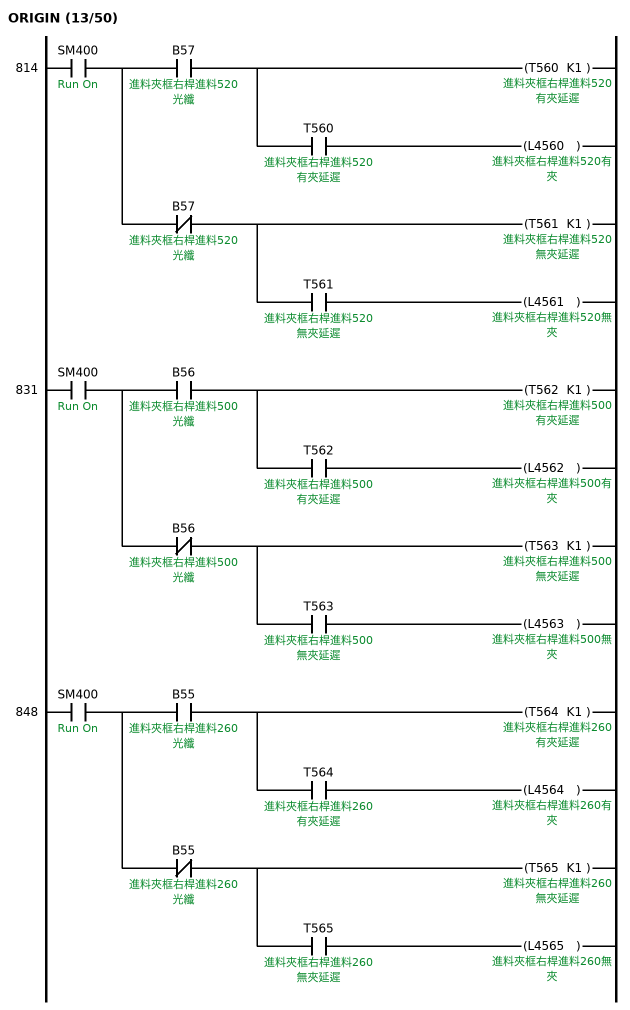
[picture p432: ladder of ORIGIN, rungs at steps 814 to 848]
814   LD      SM400  ; Run On
      MPS
      AND     B57  ; 進料夾框右桿進料520 光纖
      OUT     T560 K1  ; 進料夾框右桿進料520 有夾延遲
      AND     T560  ; 進料夾框右桿進料520 有夾延遲
      OUT     L4560  ; 進料夾框右桿進料520有夾
      MPP
      ANI     B57  ; 進料夾框右桿進料520 光纖
      OUT     T561 K1  ; 進料夾框右桿進料520 無夾延遲
      AND     T561  ; 進料夾框右桿進料520 無夾延遲
      OUT     L4561  ; 進料夾框右桿進料520無夾
831   LD      SM400  ; Run On
      MPS
      AND     B56  ; 進料夾框右桿進料500 光纖
      OUT     T562 K1  ; 進料夾框右桿進料500 有夾延遲
      AND     T562  ; 進料夾框右桿進料500 有夾延遲
      OUT     L4562  ; 進料夾框右桿進料500有夾
      MPP
      ANI     B56  ; 進料夾框右桿進料500 光纖
      OUT     T563 K1  ; 進料夾框右桿進料500 無夾延遲
      AND     T563  ; 進料夾框右桿進料500 無夾延遲
      OUT     L4563  ; 進料夾框右桿進料500無夾
848   LD      SM400  ; Run On
      MPS
      AND     B55  ; 進料夾框右桿進料260 光纖
      OUT     T564 K1  ; 進料夾框右桿進料260 有夾延遲
      AND     T564  ; 進料夾框右桿進料260 有夾延遲
      OUT     L4564  ; 進料夾框右桿進料260有夾
      MPP
      ANI     B55  ; 進料夾框右桿進料260 光纖
      OUT     T565 K1  ; 進料夾框右桿進料260 無夾延遲
      AND     T565  ; 進料夾框右桿進料260 無夾延遲
      OUT     L4565  ; 進料夾框右桿進料260無夾
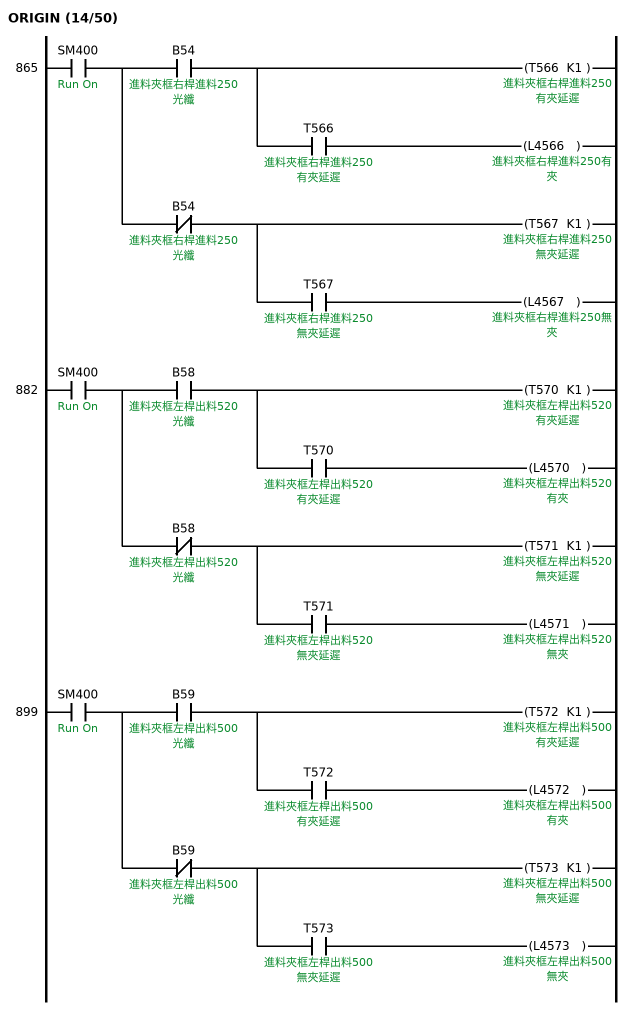
865   LD      SM400  ; Run On
      MPS
      AND     B54  ; 進料夾框右桿進料250 光纖
      OUT     T566 K1  ; 進料夾框右桿進料250 有夾延遲
      AND     T566  ; 進料夾框右桿進料250 有夾延遲
      OUT     L4566  ; 進料夾框右桿進料250有夾
      MPP
      ANI     B54  ; 進料夾框右桿進料250 光纖
      OUT     T567 K1  ; 進料夾框右桿進料250 無夾延遲
      AND     T567  ; 進料夾框右桿進料250 無夾延遲
      OUT     L4567  ; 進料夾框右桿進料250無夾
882   LD      SM400  ; Run On
      MPS
      AND     B58  ; 進料夾框左桿出料520 光纖
      OUT     T570 K1  ; 進料夾框左桿出料520 有夾延遲
      AND     T570  ; 進料夾框左桿出料520 有夾延遲
      OUT     L4570  ; 進料夾框左桿出料520 有夾
      MPP
      ANI     B58  ; 進料夾框左桿出料520 光纖
      OUT     T571 K1  ; 進料夾框左桿出料520 無夾延遲
      AND     T571  ; 進料夾框左桿出料520 無夾延遲
      OUT     L4571  ; 進料夾框左桿出料520 無夾
899   LD      SM400  ; Run On
      MPS
      AND     B59  ; 進料夾框左桿出料500 光纖
      OUT     T572 K1  ; 進料夾框左桿出料500 有夾延遲
      AND     T572  ; 進料夾框左桿出料500 有夾延遲
      OUT     L4572  ; 進料夾框左桿出料500 有夾
      MPP
      ANI     B59  ; 進料夾框左桿出料500 光纖
      OUT     T573 K1  ; 進料夾框左桿出料500 無夾延遲
      AND     T573  ; 進料夾框左桿出料500 無夾延遲
      OUT     L4573  ; 進料夾框左桿出料500 無夾
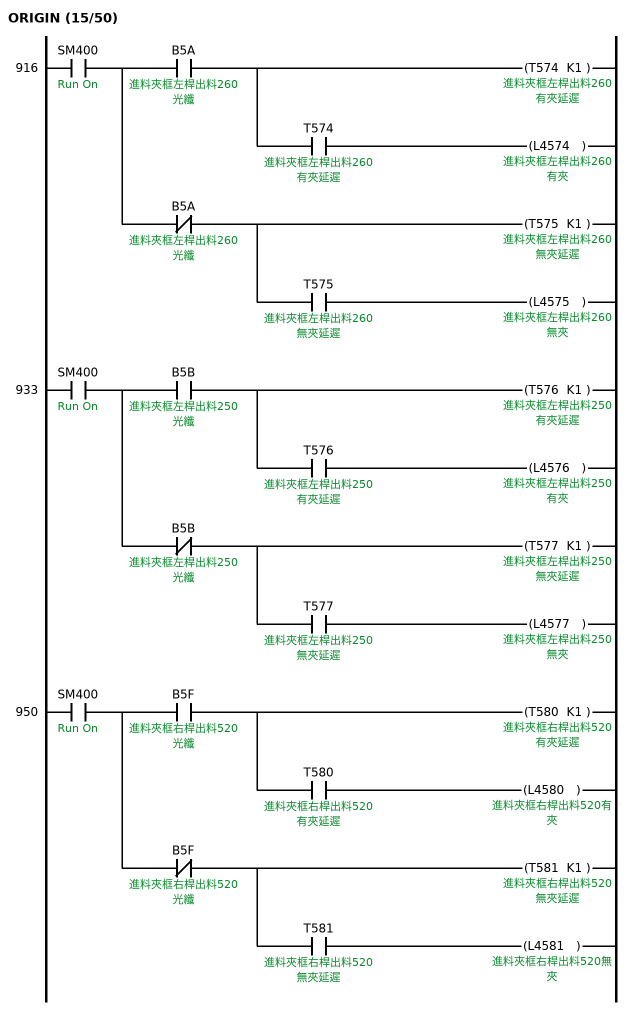
916   LD      SM400  ; Run On
      MPS
      AND     B5A  ; 進料夾框左桿出料260 光纖
      OUT     T574 K1  ; 進料夾框左桿出料260 有夾延遲
      AND     T574  ; 進料夾框左桿出料260 有夾延遲
      OUT     L4574  ; 進料夾框左桿出料260 有夾
      MPP
      ANI     B5A  ; 進料夾框左桿出料260 光纖
      OUT     T575 K1  ; 進料夾框左桿出料260 無夾延遲
      AND     T575  ; 進料夾框左桿出料260 無夾延遲
      OUT     L4575  ; 進料夾框左桿出料260 無夾
933   LD      SM400  ; Run On
      MPS
      AND     B5B  ; 進料夾框左桿出料250 光纖
      OUT     T576 K1  ; 進料夾框左桿出料250 有夾延遲
      AND     T576  ; 進料夾框左桿出料250 有夾延遲
      OUT     L4576  ; 進料夾框左桿出料250 有夾
      MPP
      ANI     B5B  ; 進料夾框左桿出料250 光纖
      OUT     T577 K1  ; 進料夾框左桿出料250 無夾延遲
      AND     T577  ; 進料夾框左桿出料250 無夾延遲
      OUT     L4577  ; 進料夾框左桿出料250 無夾
950   LD      SM400  ; Run On
      MPS
      AND     B5F  ; 進料夾框右桿出料520 光纖
      OUT     T580 K1  ; 進料夾框右桿出料520 有夾延遲
      AND     T580  ; 進料夾框右桿出料520 有夾延遲
      OUT     L4580  ; 進料夾框右桿出料520有夾
      MPP
      ANI     B5F  ; 進料夾框右桿出料520 光纖
      OUT     T581 K1  ; 進料夾框右桿出料520 無夾延遲
      AND     T581  ; 進料夾框右桿出料520 無夾延遲
      OUT     L4581  ; 進料夾框右桿出料520無夾
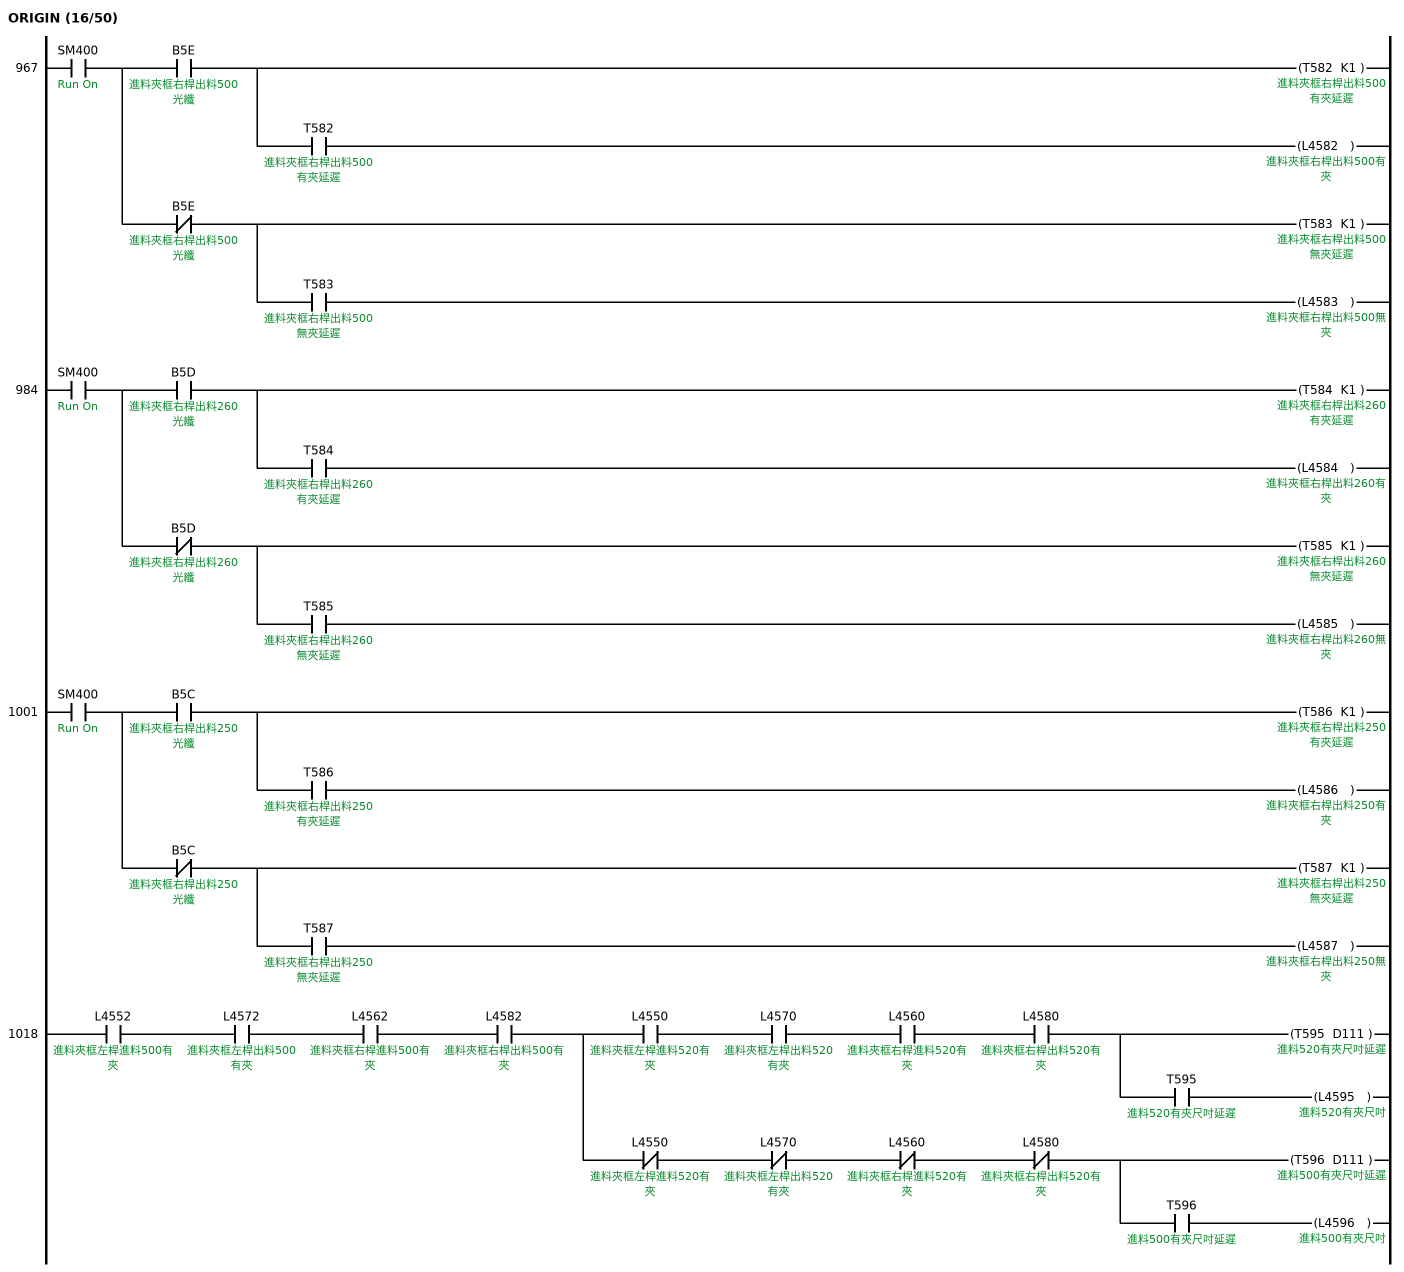
967   LD      SM400  ; Run On
      MPS
      AND     B5E  ; 進料夾框右桿出料500 光纖
      OUT     T582 K1  ; 進料夾框右桿出料500 有夾延遲
      AND     T582  ; 進料夾框右桿出料500 有夾延遲
      OUT     L4582  ; 進料夾框右桿出料500有夾
      MPP
      ANI     B5E  ; 進料夾框右桿出料500 光纖
      OUT     T583 K1  ; 進料夾框右桿出料500 無夾延遲
      AND     T583  ; 進料夾框右桿出料500 無夾延遲
      OUT     L4583  ; 進料夾框右桿出料500無夾
984   LD      SM400  ; Run On
      MPS
      AND     B5D  ; 進料夾框右桿出料260 光纖
      OUT     T584 K1  ; 進料夾框右桿出料260 有夾延遲
      AND     T584  ; 進料夾框右桿出料260 有夾延遲
      OUT     L4584  ; 進料夾框右桿出料260有夾
      MPP
      ANI     B5D  ; 進料夾框右桿出料260 光纖
      OUT     T585 K1  ; 進料夾框右桿出料260 無夾延遲
      AND     T585  ; 進料夾框右桿出料260 無夾延遲
      OUT     L4585  ; 進料夾框右桿出料260無夾
1001  LD      SM400  ; Run On
      MPS
      AND     B5C  ; 進料夾框右桿出料250 光纖
      OUT     T586 K1  ; 進料夾框右桿出料250 有夾延遲
      AND     T586  ; 進料夾框右桿出料250 有夾延遲
      OUT     L4586  ; 進料夾框右桿出料250有夾
      MPP
      ANI     B5C  ; 進料夾框右桿出料250 光纖
      OUT     T587 K1  ; 進料夾框右桿出料250 無夾延遲
      AND     T587  ; 進料夾框右桿出料250 無夾延遲
      OUT     L4587  ; 進料夾框右桿出料250無夾
1018  LD      L4552  ; 進料夾框左桿進料500有夾
      AND     L4572  ; 進料夾框左桿出料500 有夾
      AND     L4562  ; 進料夾框右桿進料500有夾
      AND     L4582  ; 進料夾框右桿出料500有夾
      MPS
      AND     L4550  ; 進料夾框左桿進料520有夾
      AND     L4570  ; 進料夾框左桿出料520 有夾
      AND     L4560  ; 進料夾框右桿進料520有夾
      AND     L4580  ; 進料夾框右桿出料520有夾
      OUT     T595 D111  ; 進料520有夾尺吋延遲
      AND     T595  ; 進料520有夾尺吋延遲
      OUT     L4595  ; 進料520有夾尺吋
      MPP
      ANI     L4550  ; 進料夾框左桿進料520有夾
      ANI     L4570  ; 進料夾框左桿出料520 有夾
      ANI     L4560  ; 進料夾框右桿進料520有夾
      ANI     L4580  ; 進料夾框右桿出料520有夾
      OUT     T596 D111  ; 進料500有夾尺吋延遲
      AND     T596  ; 進料500有夾尺吋延遲
      OUT     L4596  ; 進料500有夾尺吋
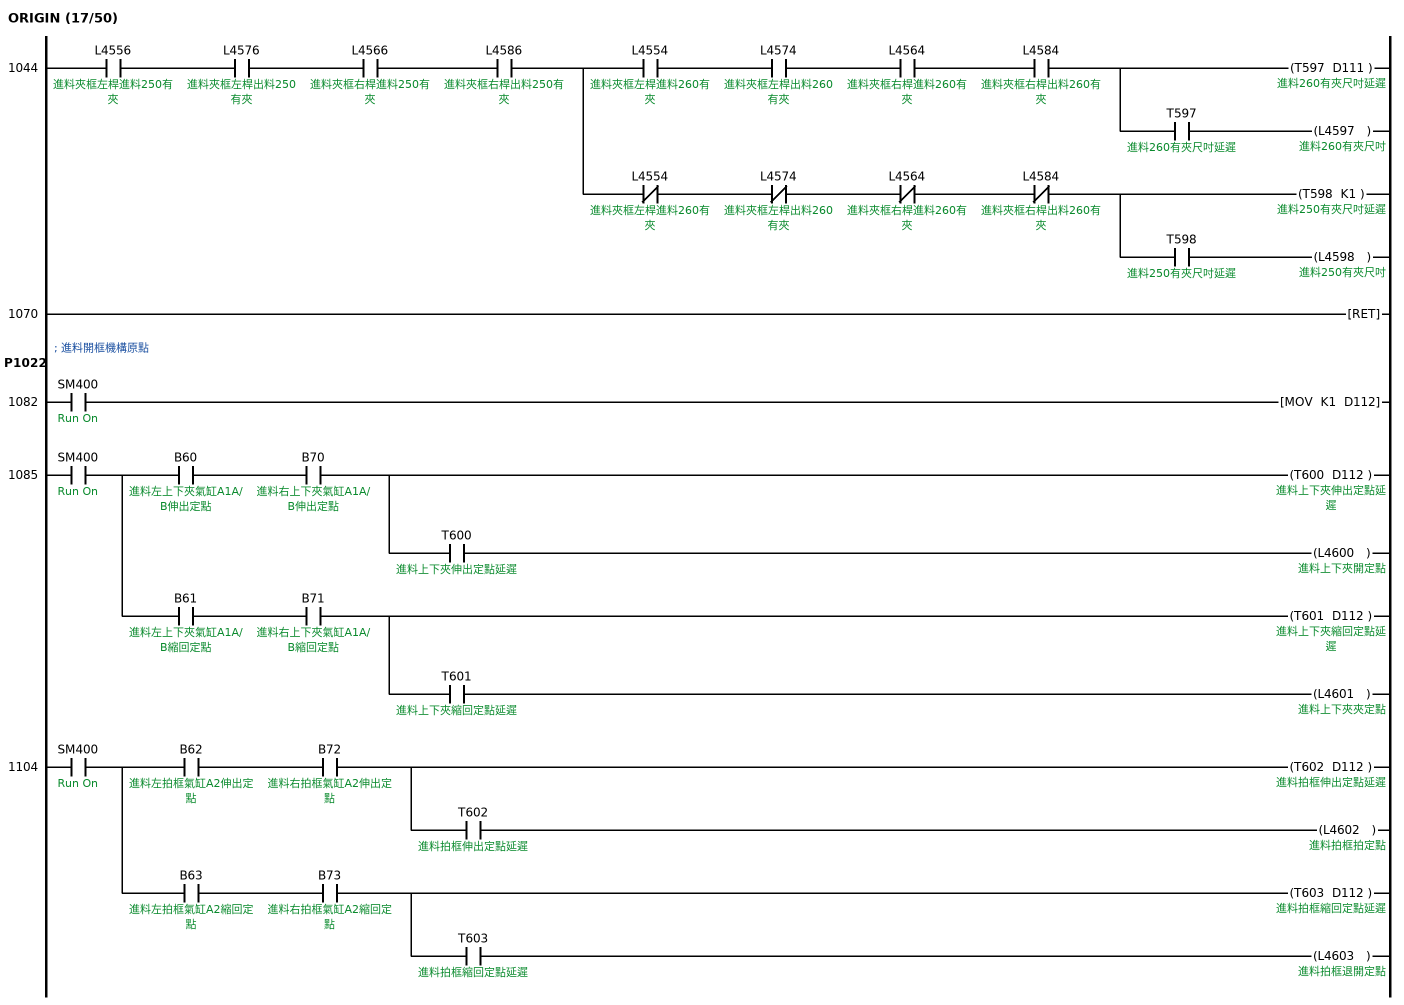
1044  LD      L4556  ; 進料夾框左桿進料250有夾
      AND     L4576  ; 進料夾框左桿出料250 有夾
      AND     L4566  ; 進料夾框右桿進料250有夾
      AND     L4586  ; 進料夾框右桿出料250有夾
      MPS
      AND     L4554  ; 進料夾框左桿進料260有夾
      AND     L4574  ; 進料夾框左桿出料260 有夾
      AND     L4564  ; 進料夾框右桿進料260有夾
      AND     L4584  ; 進料夾框右桿出料260有夾
      OUT     T597 D111  ; 進料260有夾尺吋延遲
      AND     T597  ; 進料260有夾尺吋延遲
      OUT     L4597  ; 進料260有夾尺吋
      MPP
      ANI     L4554  ; 進料夾框左桿進料260有夾
      ANI     L4574  ; 進料夾框左桿出料260 有夾
      ANI     L4564  ; 進料夾框右桿進料260有夾
      ANI     L4584  ; 進料夾框右桿出料260有夾
      OUT     T598 K1  ; 進料250有夾尺吋延遲
      AND     T598  ; 進料250有夾尺吋延遲
      OUT     L4598  ; 進料250有夾尺吋
1070  RET
; 進料開框機構原點
      P1022
1082  LD      SM400  ; Run On
      MOV     K1 D112
1085  LD      SM400  ; Run On
      MPS
      AND     B60  ; 進料左上下夾氣缸A1A/B伸出定點
      AND     B70  ; 進料右上下夾氣缸A1A/B伸出定點
      OUT     T600 D112  ; 進料上下夾伸出定點延遲
      AND     T600  ; 進料上下夾伸出定點延遲
      OUT     L4600  ; 進料上下夾開定點
      MPP
      AND     B61  ; 進料左上下夾氣缸A1A/B縮回定點
      AND     B71  ; 進料右上下夾氣缸A1A/B縮回定點
      OUT     T601 D112  ; 進料上下夾縮回定點延遲
      AND     T601  ; 進料上下夾縮回定點延遲
      OUT     L4601  ; 進料上下夾夾定點
1104  LD      SM400  ; Run On
      MPS
      AND     B62  ; 進料左拍框氣缸A2伸出定點
      AND     B72  ; 進料右拍框氣缸A2伸出定點
      OUT     T602 D112  ; 進料拍框伸出定點延遲
      AND     T602  ; 進料拍框伸出定點延遲
      OUT     L4602  ; 進料拍框拍定點
      MPP
      AND     B63  ; 進料左拍框氣缸A2縮回定點
      AND     B73  ; 進料右拍框氣缸A2縮回定點
      OUT     T603 D112  ; 進料拍框縮回定點延遲
      AND     T603  ; 進料拍框縮回定點延遲
      OUT     L4603  ; 進料拍框退開定點
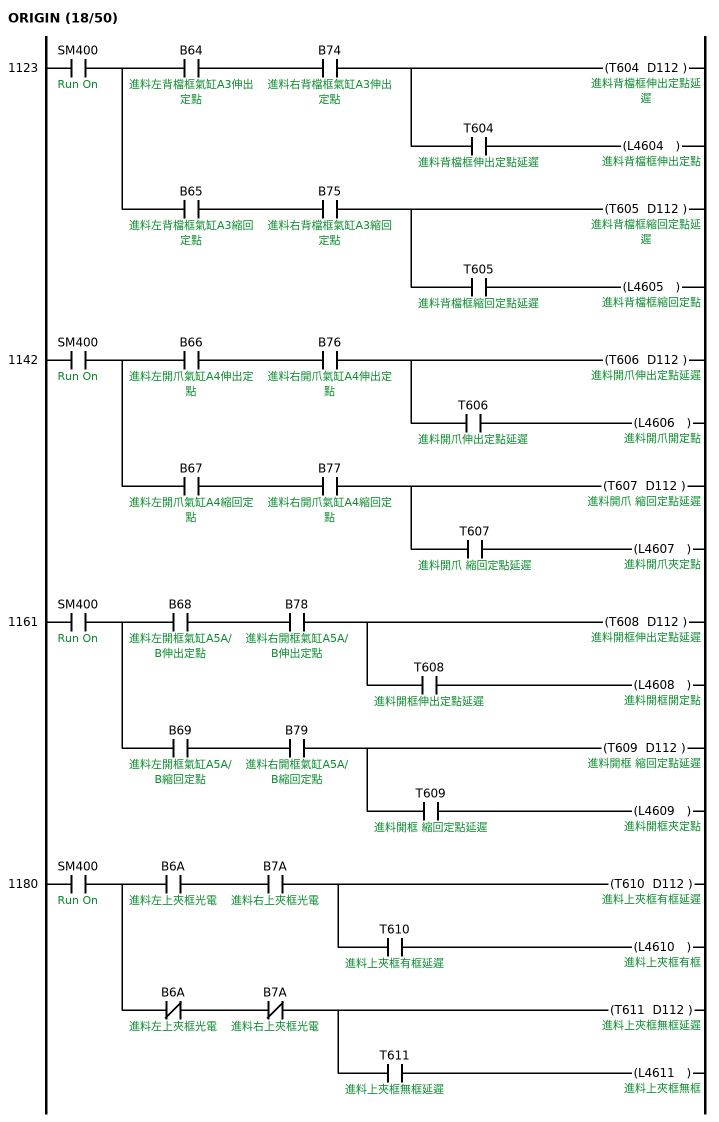
1123  LD      SM400  ; Run On
      MPS
      AND     B64  ; 進料左背檔框氣缸A3伸出定點
      AND     B74  ; 進料右背檔框氣缸A3伸出定點
      OUT     T604 D112  ; 進料背檔框伸出定點延遲
      AND     T604  ; 進料背檔框伸出定點延遲
      OUT     L4604  ; 進料背檔框伸出定點
      MPP
      AND     B65  ; 進料左背檔框氣缸A3縮回定點
      AND     B75  ; 進料右背檔框氣缸A3縮回定點
      OUT     T605 D112  ; 進料背檔框縮回定點延遲
      AND     T605  ; 進料背檔框縮回定點延遲
      OUT     L4605  ; 進料背檔框縮回定點
1142  LD      SM400  ; Run On
      MPS
      AND     B66  ; 進料左開爪氣缸A4伸出定點
      AND     B76  ; 進料右開爪氣缸A4伸出定點
      OUT     T606 D112  ; 進料開爪伸出定點延遲
      AND     T606  ; 進料開爪伸出定點延遲
      OUT     L4606  ; 進料開爪開定點
      MPP
      AND     B67  ; 進料左開爪氣缸A4縮回定點
      AND     B77  ; 進料右開爪氣缸A4縮回定點
      OUT     T607 D112  ; 進料開爪 縮回定點延遲
      AND     T607  ; 進料開爪 縮回定點延遲
      OUT     L4607  ; 進料開爪夾定點
1161  LD      SM400  ; Run On
      MPS
      AND     B68  ; 進料左開框氣缸A5A/B伸出定點
      AND     B78  ; 進料右開框氣缸A5A/B伸出定點
      OUT     T608 D112  ; 進料開框伸出定點延遲
      AND     T608  ; 進料開框伸出定點延遲
      OUT     L4608  ; 進料開框開定點
      MPP
      AND     B69  ; 進料左開框氣缸A5A/B縮回定點
      AND     B79  ; 進料右開框氣缸A5A/B縮回定點
      OUT     T609 D112  ; 進料開框 縮回定點延遲
      AND     T609  ; 進料開框 縮回定點延遲
      OUT     L4609  ; 進料開框夾定點
1180  LD      SM400  ; Run On
      MPS
      AND     B6A  ; 進料左上夾框光電
      AND     B7A  ; 進料右上夾框光電
      OUT     T610 D112  ; 進料上夾框有框延遲
      AND     T610  ; 進料上夾框有框延遲
      OUT     L4610  ; 進料上夾框有框
      MPP
      ANI     B6A  ; 進料左上夾框光電
      ANI     B7A  ; 進料右上夾框光電
      OUT     T611 D112  ; 進料上夾框無框延遲
      AND     T611  ; 進料上夾框無框延遲
      OUT     L4611  ; 進料上夾框無框
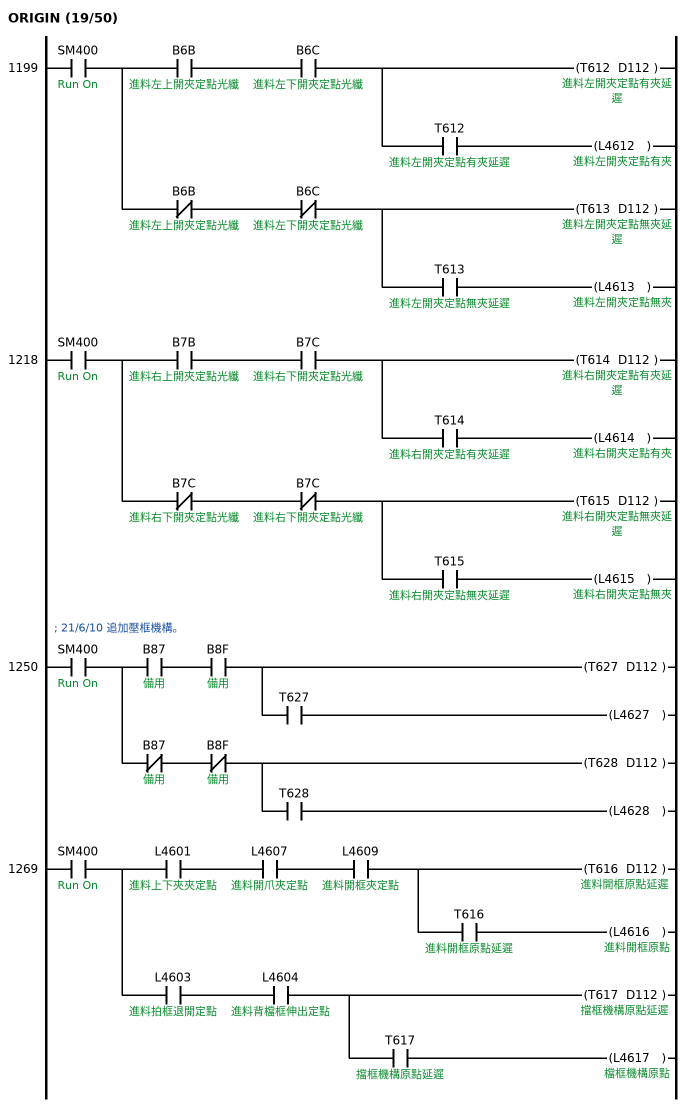
1199  LD      SM400  ; Run On
      MPS
      AND     B6B  ; 進料左上開夾定點光纖
      AND     B6C  ; 進料左下開夾定點光纖
      OUT     T612 D112  ; 進料左開夾定點有夾延遲
      AND     T612  ; 進料左開夾定點有夾延遲
      OUT     L4612  ; 進料左開夾定點有夾
      MPP
      ANI     B6B  ; 進料左上開夾定點光纖
      ANI     B6C  ; 進料左下開夾定點光纖
      OUT     T613 D112  ; 進料左開夾定點無夾延遲
      AND     T613  ; 進料左開夾定點無夾延遲
      OUT     L4613  ; 進料左開夾定點無夾
1218  LD      SM400  ; Run On
      MPS
      AND     B7B  ; 進料右上開夾定點光纖
      AND     B7C  ; 進料右下開夾定點光纖
      OUT     T614 D112  ; 進料右開夾定點有夾延遲
      AND     T614  ; 進料右開夾定點有夾延遲
      OUT     L4614  ; 進料右開夾定點有夾
      MPP
      ANI     B7C  ; 進料右下開夾定點光纖
      ANI     B7C  ; 進料右下開夾定點光纖
      OUT     T615 D112  ; 進料右開夾定點無夾延遲
      AND     T615  ; 進料右開夾定點無夾延遲
      OUT     L4615  ; 進料右開夾定點無夾
; 21/6/10 追加壓框機構。
1250  LD      SM400  ; Run On
      MPS
      AND     B87  ; 備用
      AND     B8F  ; 備用
      OUT     T627 D112
      AND     T627
      OUT     L4627
      MPP
      ANI     B87  ; 備用
      ANI     B8F  ; 備用
      OUT     T628 D112
      AND     T628
      OUT     L4628
1269  LD      SM400  ; Run On
      MPS
      AND     L4601  ; 進料上下夾夾定點
      AND     L4607  ; 進料開爪夾定點
      AND     L4609  ; 進料開框夾定點
      OUT     T616 D112  ; 進料開框原點延遲
      AND     T616  ; 進料開框原點延遲
      OUT     L4616  ; 進料開框原點
      MPP
      AND     L4603  ; 進料拍框退開定點
      AND     L4604  ; 進料背檔框伸出定點
      OUT     T617 D112  ; 擋框機構原點延遲
      AND     T617  ; 擋框機構原點延遲
      OUT     L4617  ; 檔框機構原點
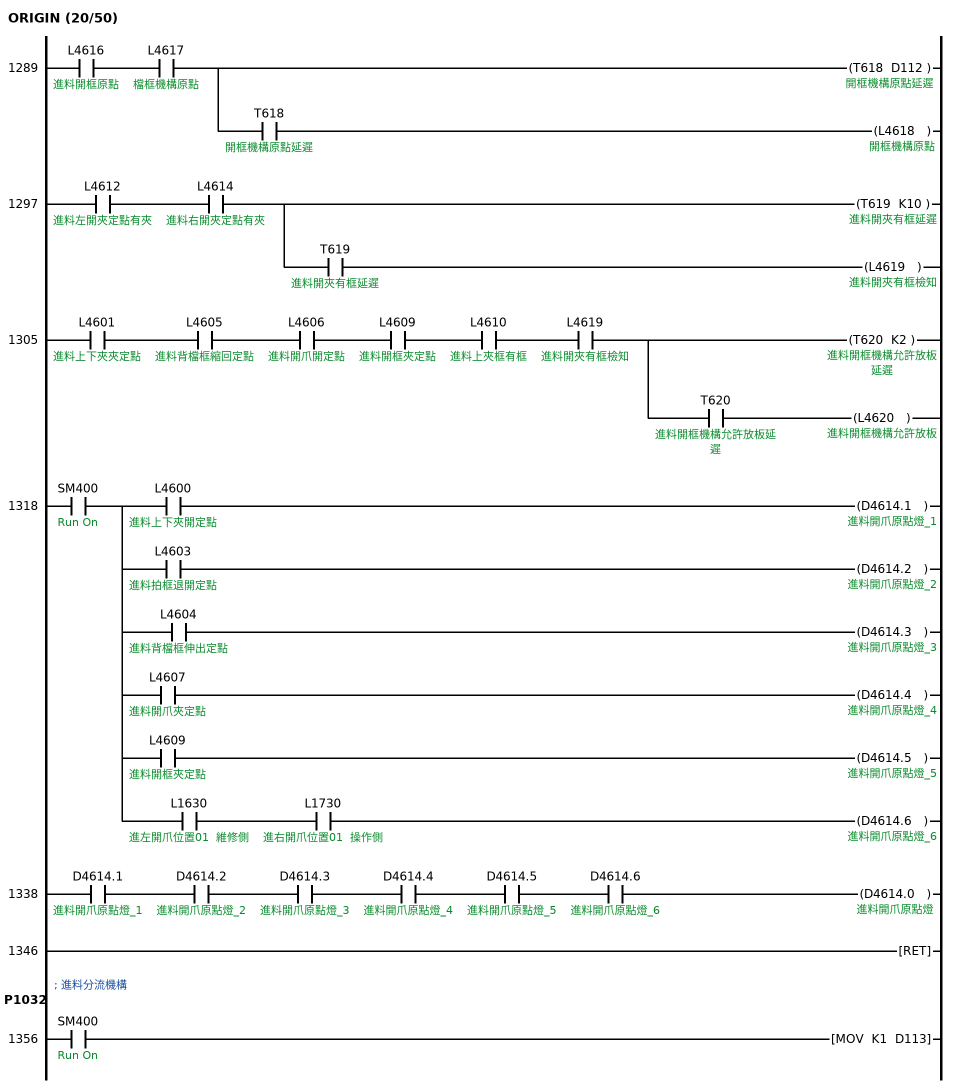
1289  LD      L4616  ; 進料開框原點
      AND     L4617  ; 檔框機構原點
      OUT     T618 D112  ; 開框機構原點延遲
      AND     T618  ; 開框機構原點延遲
      OUT     L4618  ; 開框機構原點
1297  LD      L4612  ; 進料左開夾定點有夾
      AND     L4614  ; 進料右開夾定點有夾
      OUT     T619 K10  ; 進料開夾有框延遲
      AND     T619  ; 進料開夾有框延遲
      OUT     L4619  ; 進料開夾有框檢知
1305  LD      L4601  ; 進料上下夾夾定點
      AND     L4605  ; 進料背檔框縮回定點
      AND     L4606  ; 進料開爪開定點
      AND     L4609  ; 進料開框夾定點
      AND     L4610  ; 進料上夾框有框
      AND     L4619  ; 進料開夾有框檢知
      OUT     T620 K2  ; 進料開框機構允許放板延遲
      AND     T620  ; 進料開框機構允許放板延遲
      OUT     L4620  ; 進料開框機構允許放板
1318  LD      SM400  ; Run On
      MPS
      AND     L4600  ; 進料上下夾開定點
      OUT     D4614.1  ; 進料開爪原點燈_1
      MRD
      AND     L4603  ; 進料拍框退開定點
      OUT     D4614.2  ; 進料開爪原點燈_2
      MRD
      AND     L4604  ; 進料背檔框伸出定點
      OUT     D4614.3  ; 進料開爪原點燈_3
      MRD
      AND     L4607  ; 進料開爪夾定點
      OUT     D4614.4  ; 進料開爪原點燈_4
      MRD
      AND     L4609  ; 進料開框夾定點
      OUT     D4614.5  ; 進料開爪原點燈_5
      MPP
      AND     L1630  ; 進左開爪位置01  維修側
      AND     L1730  ; 進右開爪位置01  操作側
      OUT     D4614.6  ; 進料開爪原點燈_6
1338  LD      D4614.1  ; 進料開爪原點燈_1
      AND     D4614.2  ; 進料開爪原點燈_2
      AND     D4614.3  ; 進料開爪原點燈_3
      AND     D4614.4  ; 進料開爪原點燈_4
      AND     D4614.5  ; 進料開爪原點燈_5
      AND     D4614.6  ; 進料開爪原點燈_6
      OUT     D4614.0  ; 進料開爪原點燈
1346  RET
; 進料分流機構
      P1032
1356  LD      SM400  ; Run On
      MOV     K1 D113
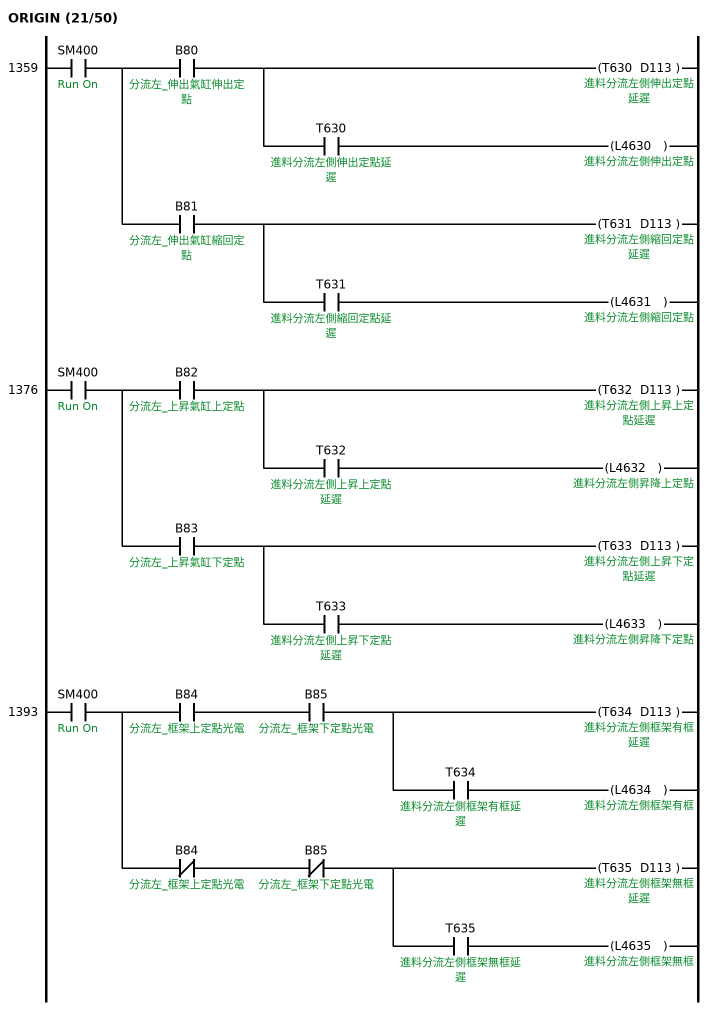
1359  LD      SM400  ; Run On
      MPS
      AND     B80  ; 分流左_伸出氣缸伸出定點
      OUT     T630 D113  ; 進料分流左側伸出定點延遲
      AND     T630  ; 進料分流左側伸出定點延遲
      OUT     L4630  ; 進料分流左側伸出定點
      MPP
      AND     B81  ; 分流左_伸出氣缸縮回定點
      OUT     T631 D113  ; 進料分流左側縮回定點延遲
      AND     T631  ; 進料分流左側縮回定點延遲
      OUT     L4631  ; 進料分流左側縮回定點
1376  LD      SM400  ; Run On
      MPS
      AND     B82  ; 分流左_上昇氣缸上定點
      OUT     T632 D113  ; 進料分流左側上昇上定點延遲
      AND     T632  ; 進料分流左側上昇上定點延遲
      OUT     L4632  ; 進料分流左側昇降上定點
      MPP
      AND     B83  ; 分流左_上昇氣缸下定點
      OUT     T633 D113  ; 進料分流左側上昇下定點延遲
      AND     T633  ; 進料分流左側上昇下定點延遲
      OUT     L4633  ; 進料分流左側昇降下定點
1393  LD      SM400  ; Run On
      MPS
      AND     B84  ; 分流左_框架上定點光電
      AND     B85  ; 分流左_框架下定點光電
      OUT     T634 D113  ; 進料分流左側框架有框延遲
      AND     T634  ; 進料分流左側框架有框延遲
      OUT     L4634  ; 進料分流左側框架有框
      MPP
      ANI     B84  ; 分流左_框架上定點光電
      ANI     B85  ; 分流左_框架下定點光電
      OUT     T635 D113  ; 進料分流左側框架無框延遲
      AND     T635  ; 進料分流左側框架無框延遲
      OUT     L4635  ; 進料分流左側框架無框
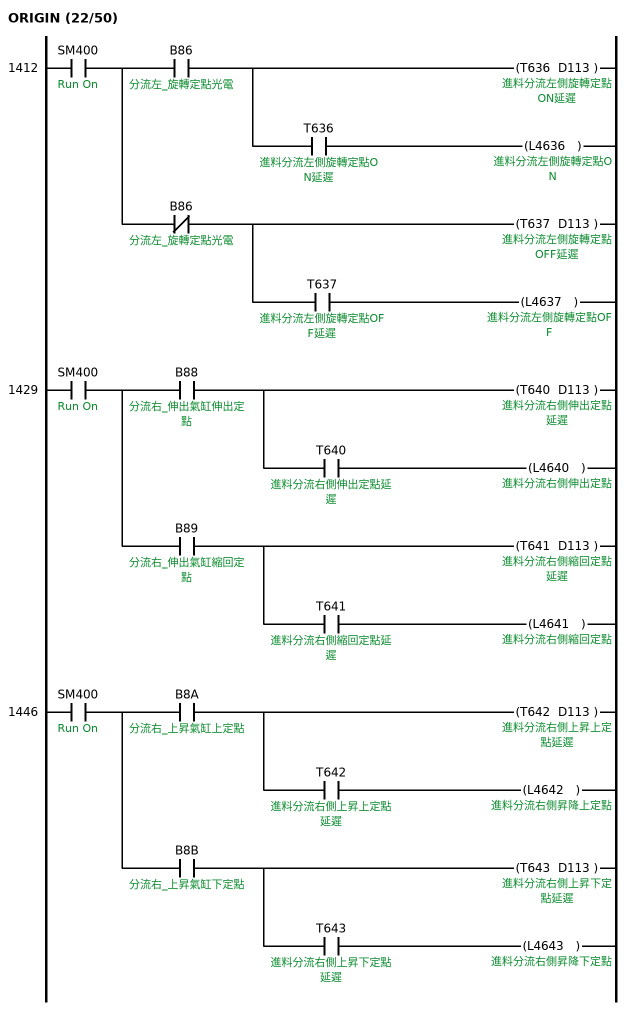
1412  LD      SM400  ; Run On
      MPS
      AND     B86  ; 分流左_旋轉定點光電
      OUT     T636 D113  ; 進料分流左側旋轉定點ON延遲
      AND     T636  ; 進料分流左側旋轉定點ON延遲
      OUT     L4636  ; 進料分流左側旋轉定點ON
      MPP
      ANI     B86  ; 分流左_旋轉定點光電
      OUT     T637 D113  ; 進料分流左側旋轉定點OFF延遲
      AND     T637  ; 進料分流左側旋轉定點OFF延遲
      OUT     L4637  ; 進料分流左側旋轉定點OFF
1429  LD      SM400  ; Run On
      MPS
      AND     B88  ; 分流右_伸出氣缸伸出定點
      OUT     T640 D113  ; 進料分流右側伸出定點延遲
      AND     T640  ; 進料分流右側伸出定點延遲
      OUT     L4640  ; 進料分流右側伸出定點
      MPP
      AND     B89  ; 分流右_伸出氣缸縮回定點
      OUT     T641 D113  ; 進料分流右側縮回定點延遲
      AND     T641  ; 進料分流右側縮回定點延遲
      OUT     L4641  ; 進料分流右側縮回定點
1446  LD      SM400  ; Run On
      MPS
      AND     B8A  ; 分流右_上昇氣缸上定點
      OUT     T642 D113  ; 進料分流右側上昇上定點延遲
      AND     T642  ; 進料分流右側上昇上定點延遲
      OUT     L4642  ; 進料分流右側昇降上定點
      MPP
      AND     B8B  ; 分流右_上昇氣缸下定點
      OUT     T643 D113  ; 進料分流右側上昇下定點延遲
      AND     T643  ; 進料分流右側上昇下定點延遲
      OUT     L4643  ; 進料分流右側昇降下定點
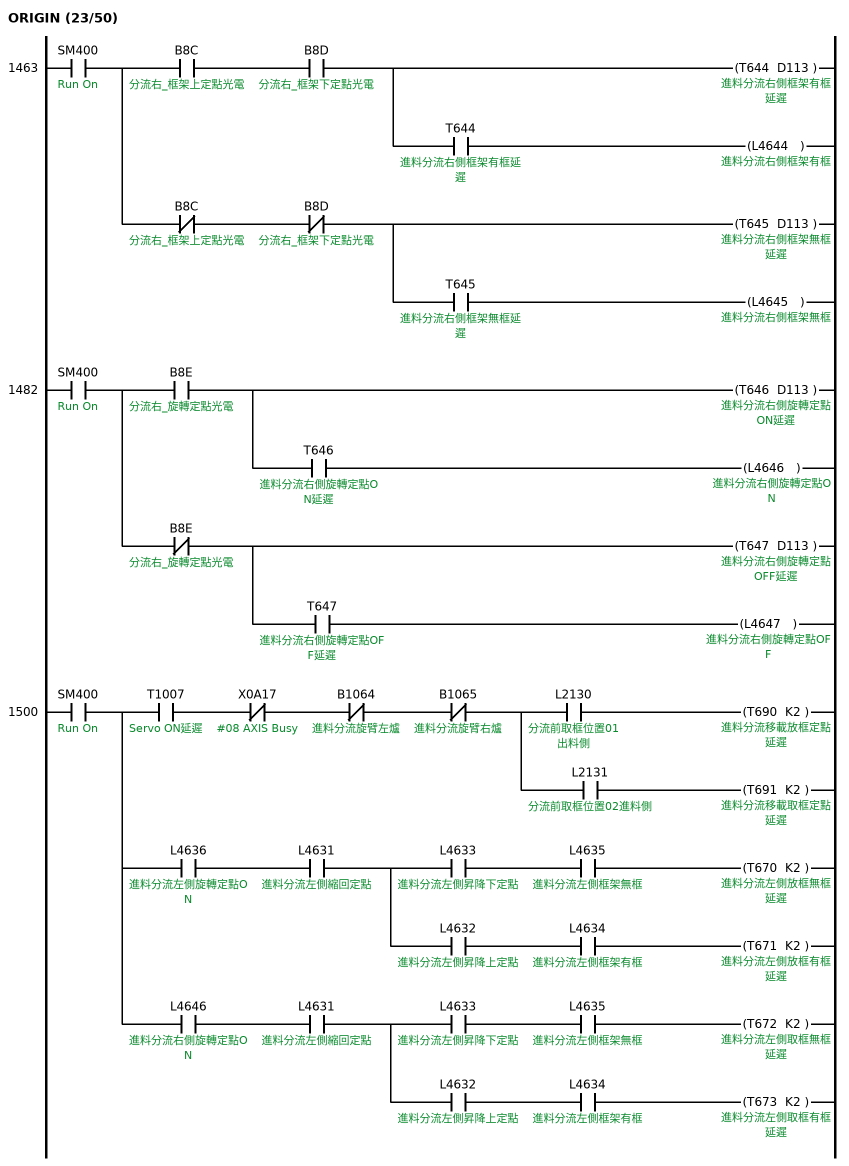
1463  LD      SM400  ; Run On
      MPS
      AND     B8C  ; 分流右_框架上定點光電
      AND     B8D  ; 分流右_框架下定點光電
      OUT     T644 D113  ; 進料分流右側框架有框延遲
      AND     T644  ; 進料分流右側框架有框延遲
      OUT     L4644  ; 進料分流右側框架有框
      MPP
      ANI     B8C  ; 分流右_框架上定點光電
      ANI     B8D  ; 分流右_框架下定點光電
      OUT     T645 D113  ; 進料分流右側框架無框延遲
      AND     T645  ; 進料分流右側框架無框延遲
      OUT     L4645  ; 進料分流右側框架無框
1482  LD      SM400  ; Run On
      MPS
      AND     B8E  ; 分流右_旋轉定點光電
      OUT     T646 D113  ; 進料分流右側旋轉定點ON延遲
      AND     T646  ; 進料分流右側旋轉定點ON延遲
      OUT     L4646  ; 進料分流右側旋轉定點ON
      MPP
      ANI     B8E  ; 分流右_旋轉定點光電
      OUT     T647 D113  ; 進料分流右側旋轉定點OFF延遲
      AND     T647  ; 進料分流右側旋轉定點OFF延遲
      OUT     L4647  ; 進料分流右側旋轉定點OFF
1500  LD      SM400  ; Run On
      MPS
      AND     T1007  ; Servo ON延遲
      ANI     X0A17  ; #08 AXIS Busy
      ANI     B1064  ; 進料分流旋臂左爐
      ANI     B1065  ; 進料分流旋臂右爐
      MPS
      AND     L2130  ; 分流前取框位置01  出料側
      OUT     T690 K2  ; 進料分流移載放框定點延遲
      MPP
      AND     L2131  ; 分流前取框位置02進料側
      OUT     T691 K2  ; 進料分流移載取框定點延遲
      MRD
      AND     L4636  ; 進料分流左側旋轉定點ON
      AND     L4631  ; 進料分流左側縮回定點
      MPS
      AND     L4633  ; 進料分流左側昇降下定點
      AND     L4635  ; 進料分流左側框架無框
      OUT     T670 K2  ; 進料分流左側放框無框延遲
      MPP
      AND     L4632  ; 進料分流左側昇降上定點
      AND     L4634  ; 進料分流左側框架有框
      OUT     T671 K2  ; 進料分流左側放框有框延遲
      MPP
      AND     L4646  ; 進料分流右側旋轉定點ON
      AND     L4631  ; 進料分流左側縮回定點
      MPS
      AND     L4633  ; 進料分流左側昇降下定點
      AND     L4635  ; 進料分流左側框架無框
      OUT     T672 K2  ; 進料分流左側取框無框延遲
      MPP
      AND     L4632  ; 進料分流左側昇降上定點
      AND     L4634  ; 進料分流左側框架有框
      OUT     T673 K2  ; 進料分流左側取框有框延遲
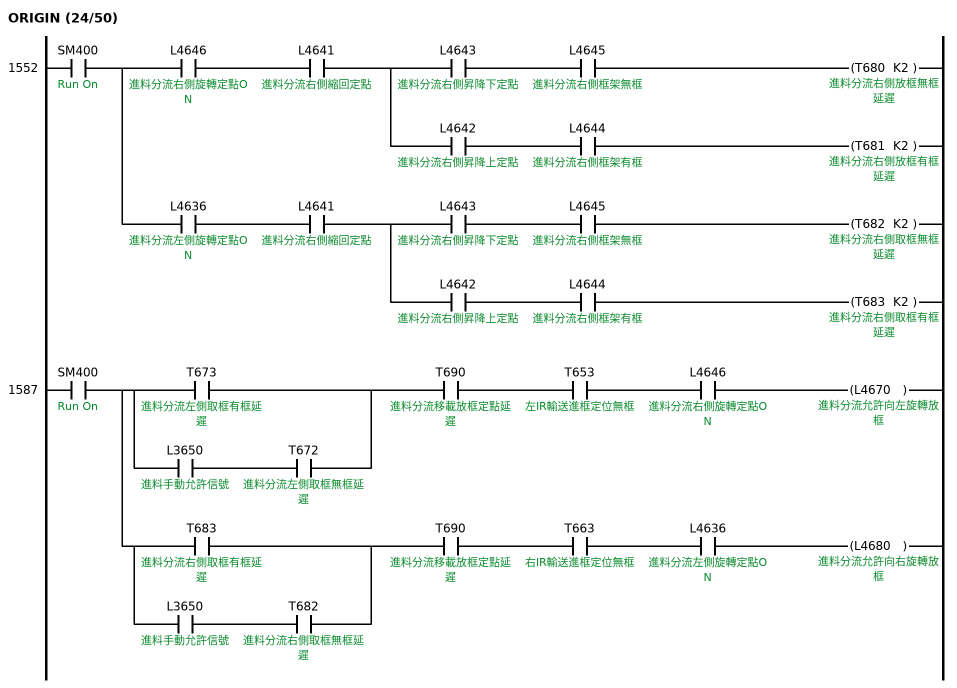
1552  LD      SM400  ; Run On
      MPS
      AND     L4646  ; 進料分流右側旋轉定點ON
      AND     L4641  ; 進料分流右側縮回定點
      MPS
      AND     L4643  ; 進料分流右側昇降下定點
      AND     L4645  ; 進料分流右側框架無框
      OUT     T680 K2  ; 進料分流右側放框無框延遲
      MPP
      AND     L4642  ; 進料分流右側昇降上定點
      AND     L4644  ; 進料分流右側框架有框
      OUT     T681 K2  ; 進料分流右側放框有框延遲
      MPP
      AND     L4636  ; 進料分流左側旋轉定點ON
      AND     L4641  ; 進料分流右側縮回定點
      MPS
      AND     L4643  ; 進料分流右側昇降下定點
      AND     L4645  ; 進料分流右側框架無框
      OUT     T682 K2  ; 進料分流右側取框無框延遲
      MPP
      AND     L4642  ; 進料分流右側昇降上定點
      AND     L4644  ; 進料分流右側框架有框
      OUT     T683 K2  ; 進料分流右側取框有框延遲
1587  LD      SM400  ; Run On
      MPS
      LD      T673  ; 進料分流左側取框有框延遲
      LD      L3650  ; 進料手動允許信號
      AND     T672  ; 進料分流左側取框無框延遲
      ORB
      ANB
      AND     T690  ; 進料分流移載放框定點延遲
      AND     T653  ; 左IR輸送進框定位無框
      AND     L4646  ; 進料分流右側旋轉定點ON
      OUT     L4670  ; 進料分流允許向左旋轉放框
      MPP
      LD      T683  ; 進料分流右側取框有框延遲
      LD      L3650  ; 進料手動允許信號
      AND     T682  ; 進料分流右側取框無框延遲
      ORB
      ANB
      AND     T690  ; 進料分流移載放框定點延遲
      AND     T663  ; 右IR輸送進框定位無框
      AND     L4636  ; 進料分流左側旋轉定點ON
      OUT     L4680  ; 進料分流允許向右旋轉放框
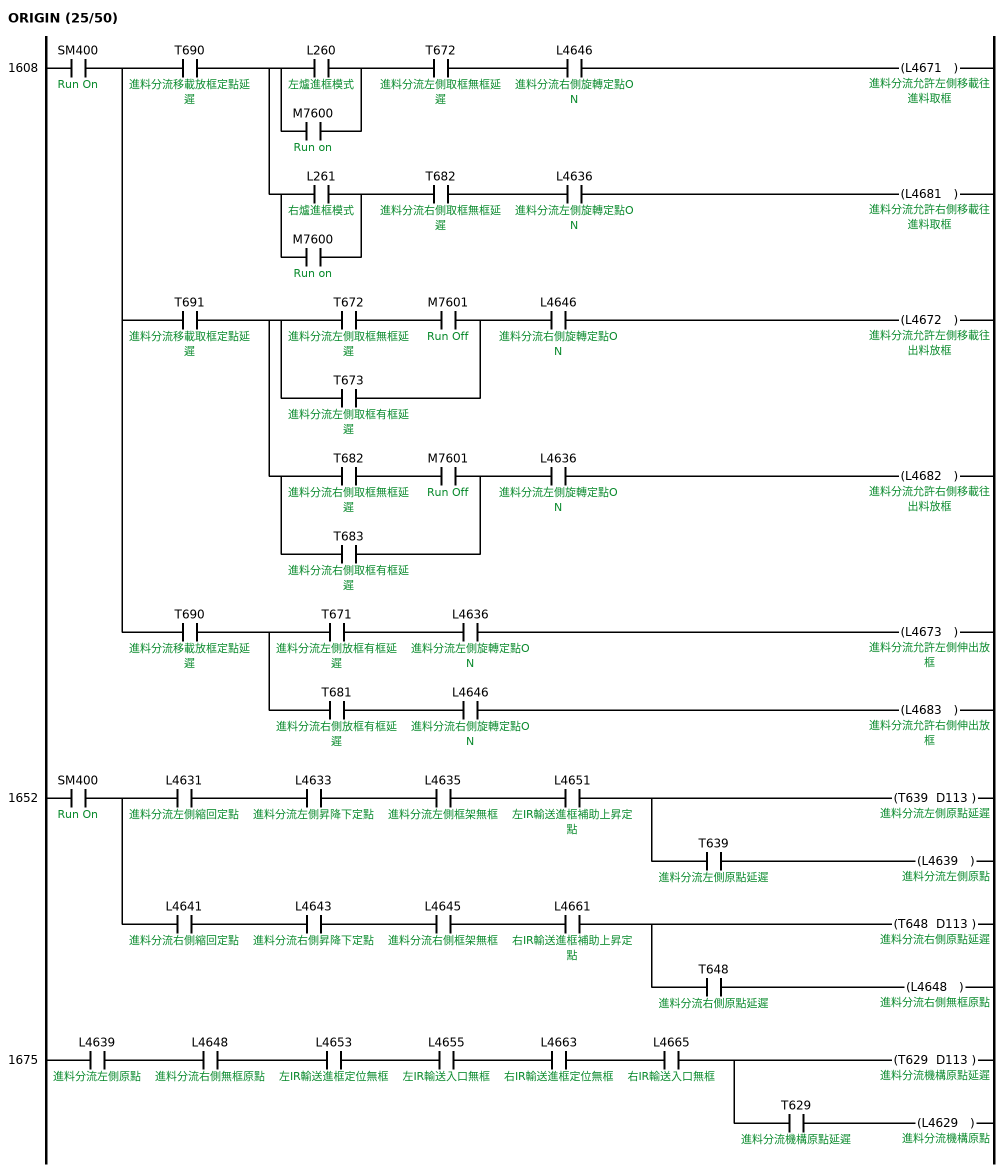
1608  LD      SM400  ; Run On
      MPS
      AND     T690  ; 進料分流移載放框定點延遲
      MPS
      LD      L260  ; 左爐進框模式
      OR      M7600  ; Run on
      ANB
      AND     T672  ; 進料分流左側取框無框延遲
      AND     L4646  ; 進料分流右側旋轉定點ON
      OUT     L4671  ; 進料分流允許左側移載往  進料取框
      MPP
      LD      L261  ; 右爐進框模式
      OR      M7600  ; Run on
      ANB
      AND     T682  ; 進料分流右側取框無框延遲
      AND     L4636  ; 進料分流左側旋轉定點ON
      OUT     L4681  ; 進料分流允許右側移載往  進料取框
      MRD
      AND     T691  ; 進料分流移載取框定點延遲
      MPS
      LD      T672  ; 進料分流左側取框無框延遲
      AND     M7601  ; Run Off
      OR      T673  ; 進料分流左側取框有框延遲
      ANB
      AND     L4646  ; 進料分流右側旋轉定點ON
      OUT     L4672  ; 進料分流允許左側移載往  出料放框
      MPP
      LD      T682  ; 進料分流右側取框無框延遲
      AND     M7601  ; Run Off
      OR      T683  ; 進料分流右側取框有框延遲
      ANB
      AND     L4636  ; 進料分流左側旋轉定點ON
      OUT     L4682  ; 進料分流允許右側移載往  出料放框
      MPP
      AND     T690  ; 進料分流移載放框定點延遲
      MPS
      AND     T671  ; 進料分流左側放框有框延遲
      AND     L4636  ; 進料分流左側旋轉定點ON
      OUT     L4673  ; 進料分流允許左側伸出放框
      MPP
      AND     T681  ; 進料分流右側放框有框延遲
      AND     L4646  ; 進料分流右側旋轉定點ON
      OUT     L4683  ; 進料分流允許右側伸出放框
1652  LD      SM400  ; Run On
      MPS
      AND     L4631  ; 進料分流左側縮回定點
      AND     L4633  ; 進料分流左側昇降下定點
      AND     L4635  ; 進料分流左側框架無框
      AND     L4651  ; 左IR輸送進框補助上昇定點
      OUT     T639 D113  ; 進料分流左側原點延遲
      AND     T639  ; 進料分流左側原點延遲
      OUT     L4639  ; 進料分流左側原點
      MPP
      AND     L4641  ; 進料分流右側縮回定點
      AND     L4643  ; 進料分流右側昇降下定點
      AND     L4645  ; 進料分流右側框架無框
      AND     L4661  ; 右IR輸送進框補助上昇定點
      OUT     T648 D113  ; 進料分流右側原點延遲
      AND     T648  ; 進料分流右側原點延遲
      OUT     L4648  ; 進料分流右側無框原點
1675  LD      L4639  ; 進料分流左側原點
      AND     L4648  ; 進料分流右側無框原點
      AND     L4653  ; 左IR輸送進框定位無框
      AND     L4655  ; 左IR輸送入口無框
      AND     L4663  ; 右IR輸送進框定位無框
      AND     L4665  ; 右IR輸送入口無框
      OUT     T629 D113  ; 進料分流機構原點延遲
      AND     T629  ; 進料分流機構原點延遲
      OUT     L4629  ; 進料分流機構原點
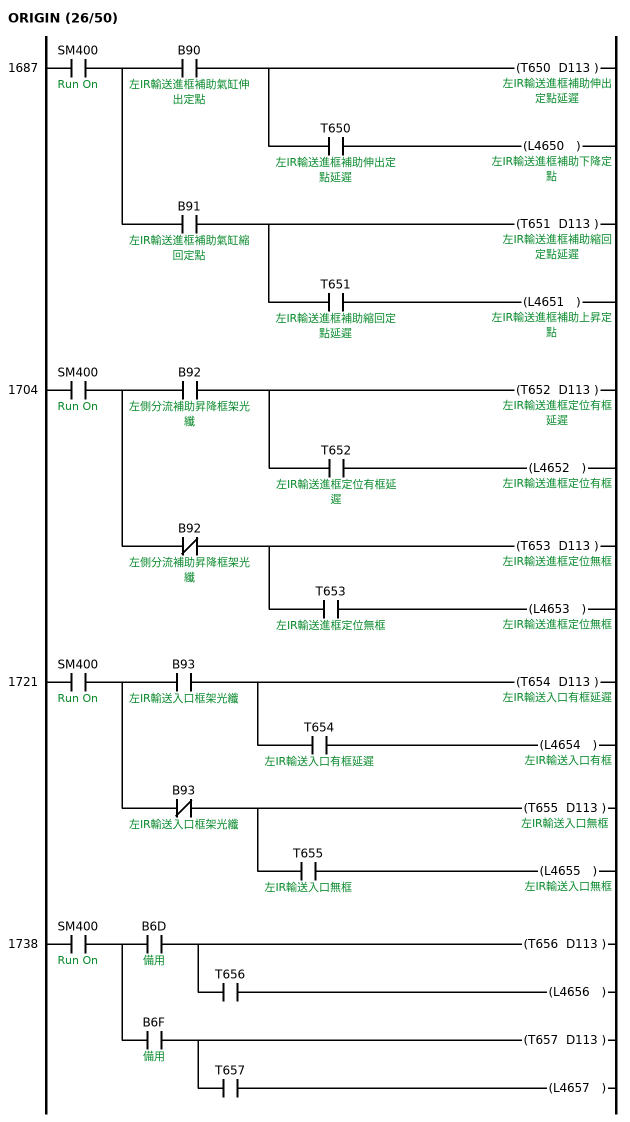
1687  LD      SM400  ; Run On
      MPS
      AND     B90  ; 左IR輸送進框補助氣缸伸出定點
      OUT     T650 D113  ; 左IR輸送進框補助伸出定點延遲
      AND     T650  ; 左IR輸送進框補助伸出定點延遲
      OUT     L4650  ; 左IR輸送進框補助下降定點
      MPP
      AND     B91  ; 左IR輸送進框補助氣缸縮回定點
      OUT     T651 D113  ; 左IR輸送進框補助縮回定點延遲
      AND     T651  ; 左IR輸送進框補助縮回定點延遲
      OUT     L4651  ; 左IR輸送進框補助上昇定點
1704  LD      SM400  ; Run On
      MPS
      AND     B92  ; 左側分流補助昇降框架光纖
      OUT     T652 D113  ; 左IR輸送進框定位有框延遲
      AND     T652  ; 左IR輸送進框定位有框延遲
      OUT     L4652  ; 左IR輸送進框定位有框
      MPP
      ANI     B92  ; 左側分流補助昇降框架光纖
      OUT     T653 D113  ; 左IR輸送進框定位無框
      AND     T653  ; 左IR輸送進框定位無框
      OUT     L4653  ; 左IR輸送進框定位無框
1721  LD      SM400  ; Run On
      MPS
      AND     B93  ; 左IR輸送入口框架光纖
      OUT     T654 D113  ; 左IR輸送入口有框延遲
      AND     T654  ; 左IR輸送入口有框延遲
      OUT     L4654  ; 左IR輸送入口有框
      MPP
      ANI     B93  ; 左IR輸送入口框架光纖
      OUT     T655 D113  ; 左IR輸送入口無框
      AND     T655  ; 左IR輸送入口無框
      OUT     L4655  ; 左IR輸送入口無框
1738  LD      SM400  ; Run On
      MPS
      AND     B6D  ; 備用
      OUT     T656 D113
      AND     T656
      OUT     L4656
      MPP
      AND     B6F  ; 備用
      OUT     T657 D113
      AND     T657
      OUT     L4657
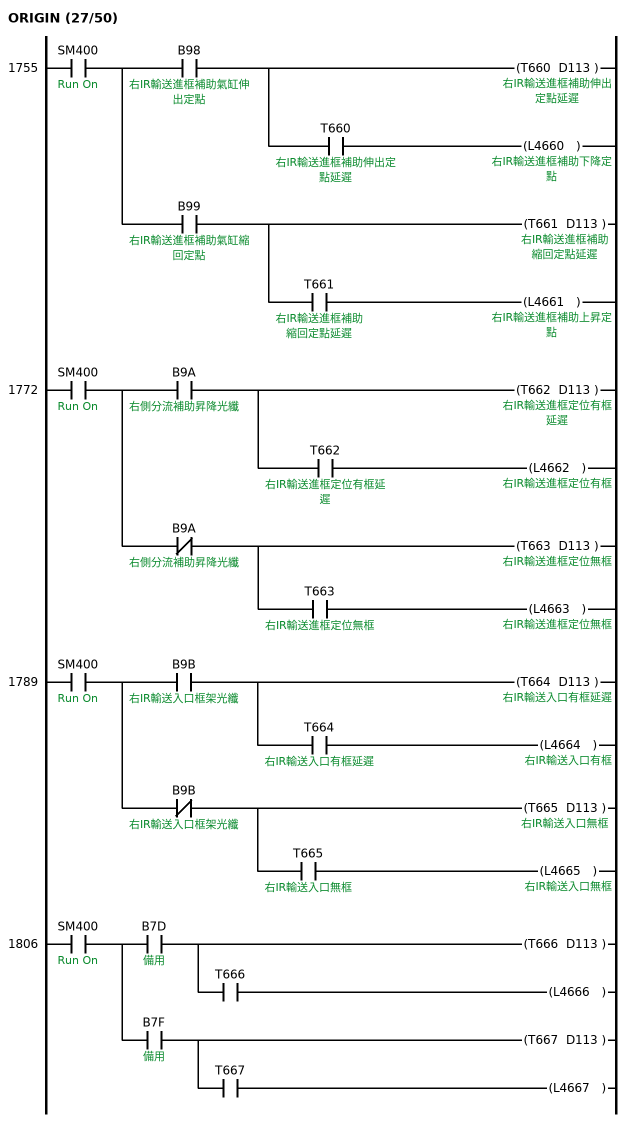
1755  LD      SM400  ; Run On
      MPS
      AND     B98  ; 右IR輸送進框補助氣缸伸出定點
      OUT     T660 D113  ; 右IR輸送進框補助伸出定點延遲
      AND     T660  ; 右IR輸送進框補助伸出定點延遲
      OUT     L4660  ; 右IR輸送進框補助下降定點
      MPP
      AND     B99  ; 右IR輸送進框補助氣缸縮回定點
      OUT     T661 D113  ; 右IR輸送進框補助 縮回定點延遲
      AND     T661  ; 右IR輸送進框補助 縮回定點延遲
      OUT     L4661  ; 右IR輸送進框補助上昇定點
1772  LD      SM400  ; Run On
      MPS
      AND     B9A  ; 右側分流補助昇降光纖
      OUT     T662 D113  ; 右IR輸送進框定位有框延遲
      AND     T662  ; 右IR輸送進框定位有框延遲
      OUT     L4662  ; 右IR輸送進框定位有框
      MPP
      ANI     B9A  ; 右側分流補助昇降光纖
      OUT     T663 D113  ; 右IR輸送進框定位無框
      AND     T663  ; 右IR輸送進框定位無框
      OUT     L4663  ; 右IR輸送進框定位無框
1789  LD      SM400  ; Run On
      MPS
      AND     B9B  ; 右IR輸送入口框架光纖
      OUT     T664 D113  ; 右IR輸送入口有框延遲
      AND     T664  ; 右IR輸送入口有框延遲
      OUT     L4664  ; 右IR輸送入口有框
      MPP
      ANI     B9B  ; 右IR輸送入口框架光纖
      OUT     T665 D113  ; 右IR輸送入口無框
      AND     T665  ; 右IR輸送入口無框
      OUT     L4665  ; 右IR輸送入口無框
1806  LD      SM400  ; Run On
      MPS
      AND     B7D  ; 備用
      OUT     T666 D113
      AND     T666
      OUT     L4666
      MPP
      AND     B7F  ; 備用
      OUT     T667 D113
      AND     T667
      OUT     L4667
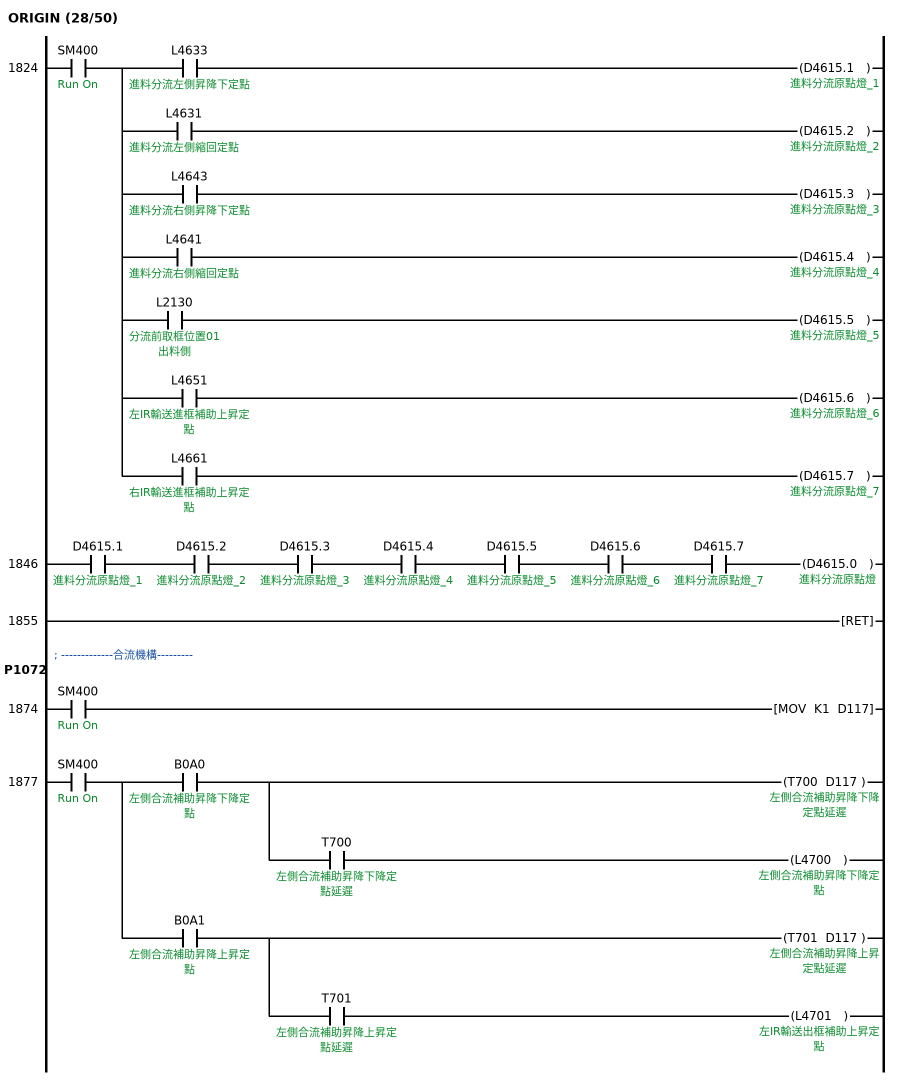
1824  LD      SM400  ; Run On
      MPS
      AND     L4633  ; 進料分流左側昇降下定點
      OUT     D4615.1  ; 進料分流原點燈_1
      MRD
      AND     L4631  ; 進料分流左側縮回定點
      OUT     D4615.2  ; 進料分流原點燈_2
      MRD
      AND     L4643  ; 進料分流右側昇降下定點
      OUT     D4615.3  ; 進料分流原點燈_3
      MRD
      AND     L4641  ; 進料分流右側縮回定點
      OUT     D4615.4  ; 進料分流原點燈_4
      MRD
      AND     L2130  ; 分流前取框位置01  出料側
      OUT     D4615.5  ; 進料分流原點燈_5
      MRD
      AND     L4651  ; 左IR輸送進框補助上昇定點
      OUT     D4615.6  ; 進料分流原點燈_6
      MPP
      AND     L4661  ; 右IR輸送進框補助上昇定點
      OUT     D4615.7  ; 進料分流原點燈_7
1846  LD      D4615.1  ; 進料分流原點燈_1
      AND     D4615.2  ; 進料分流原點燈_2
      AND     D4615.3  ; 進料分流原點燈_3
      AND     D4615.4  ; 進料分流原點燈_4
      AND     D4615.5  ; 進料分流原點燈_5
      AND     D4615.6  ; 進料分流原點燈_6
      AND     D4615.7  ; 進料分流原點燈_7
      OUT     D4615.0  ; 進料分流原點燈
1855  RET
; -------------合流機構---------
      P1072
1874  LD      SM400  ; Run On
      MOV     K1 D117
1877  LD      SM400  ; Run On
      MPS
      AND     B0A0  ; 左側合流補助昇降下降定點
      OUT     T700 D117  ; 左側合流補助昇降下降定點延遲
      AND     T700  ; 左側合流補助昇降下降定點延遲
      OUT     L4700  ; 左側合流補助昇降下降定點
      MPP
      AND     B0A1  ; 左側合流補助昇降上昇定點
      OUT     T701 D117  ; 左側合流補助昇降上昇定點延遲
      AND     T701  ; 左側合流補助昇降上昇定點延遲
      OUT     L4701  ; 左IR輸送出框補助上昇定點
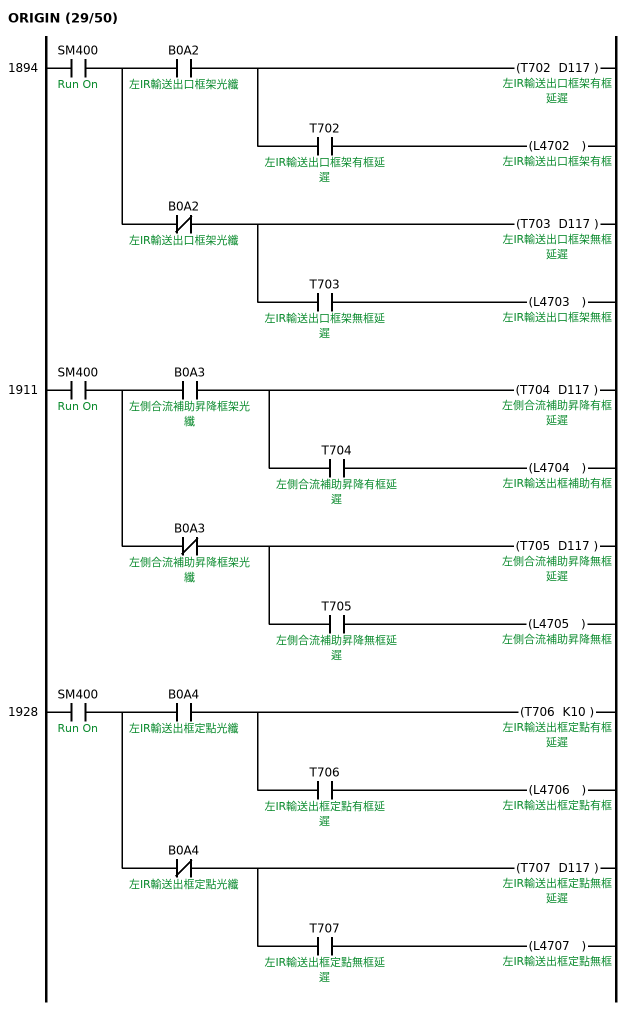
1894  LD      SM400  ; Run On
      MPS
      AND     B0A2  ; 左IR輸送出口框架光纖
      OUT     T702 D117  ; 左IR輸送出口框架有框延遲
      AND     T702  ; 左IR輸送出口框架有框延遲
      OUT     L4702  ; 左IR輸送出口框架有框
      MPP
      ANI     B0A2  ; 左IR輸送出口框架光纖
      OUT     T703 D117  ; 左IR輸送出口框架無框延遲
      AND     T703  ; 左IR輸送出口框架無框延遲
      OUT     L4703  ; 左IR輸送出口框架無框
1911  LD      SM400  ; Run On
      MPS
      AND     B0A3  ; 左側合流補助昇降框架光纖
      OUT     T704 D117  ; 左側合流補助昇降有框延遲
      AND     T704  ; 左側合流補助昇降有框延遲
      OUT     L4704  ; 左IR輸送出框補助有框
      MPP
      ANI     B0A3  ; 左側合流補助昇降框架光纖
      OUT     T705 D117  ; 左側合流補助昇降無框延遲
      AND     T705  ; 左側合流補助昇降無框延遲
      OUT     L4705  ; 左側合流補助昇降無框
1928  LD      SM400  ; Run On
      MPS
      AND     B0A4  ; 左IR輸送出框定點光纖
      OUT     T706 K10  ; 左IR輸送出框定點有框延遲
      AND     T706  ; 左IR輸送出框定點有框延遲
      OUT     L4706  ; 左IR輸送出框定點有框
      MPP
      ANI     B0A4  ; 左IR輸送出框定點光纖
      OUT     T707 D117  ; 左IR輸送出框定點無框延遲
      AND     T707  ; 左IR輸送出框定點無框延遲
      OUT     L4707  ; 左IR輸送出框定點無框
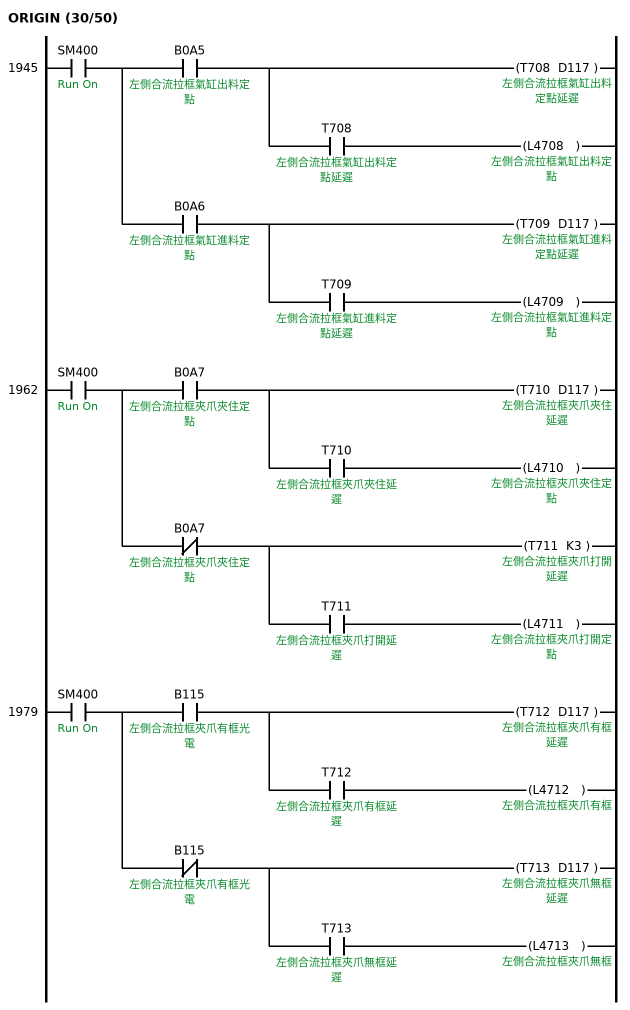
1945  LD      SM400  ; Run On
      MPS
      AND     B0A5  ; 左側合流拉框氣缸出料定點
      OUT     T708 D117  ; 左側合流拉框氣缸出料定點延遲
      AND     T708  ; 左側合流拉框氣缸出料定點延遲
      OUT     L4708  ; 左側合流拉框氣缸出料定點
      MPP
      AND     B0A6  ; 左側合流拉框氣缸進料定點
      OUT     T709 D117  ; 左側合流拉框氣缸進料定點延遲
      AND     T709  ; 左側合流拉框氣缸進料定點延遲
      OUT     L4709  ; 左側合流拉框氣缸進料定點
1962  LD      SM400  ; Run On
      MPS
      AND     B0A7  ; 左側合流拉框夾爪夾住定點
      OUT     T710 D117  ; 左側合流拉框夾爪夾住延遲
      AND     T710  ; 左側合流拉框夾爪夾住延遲
      OUT     L4710  ; 左側合流拉框夾爪夾住定點
      MPP
      ANI     B0A7  ; 左側合流拉框夾爪夾住定點
      OUT     T711 K3  ; 左側合流拉框夾爪打開延遲
      AND     T711  ; 左側合流拉框夾爪打開延遲
      OUT     L4711  ; 左側合流拉框夾爪打開定點
1979  LD      SM400  ; Run On
      MPS
      AND     B115  ; 左側合流拉框夾爪有框光電
      OUT     T712 D117  ; 左側合流拉框夾爪有框延遲
      AND     T712  ; 左側合流拉框夾爪有框延遲
      OUT     L4712  ; 左側合流拉框夾爪有框
      MPP
      ANI     B115  ; 左側合流拉框夾爪有框光電
      OUT     T713 D117  ; 左側合流拉框夾爪無框延遲
      AND     T713  ; 左側合流拉框夾爪無框延遲
      OUT     L4713  ; 左側合流拉框夾爪無框
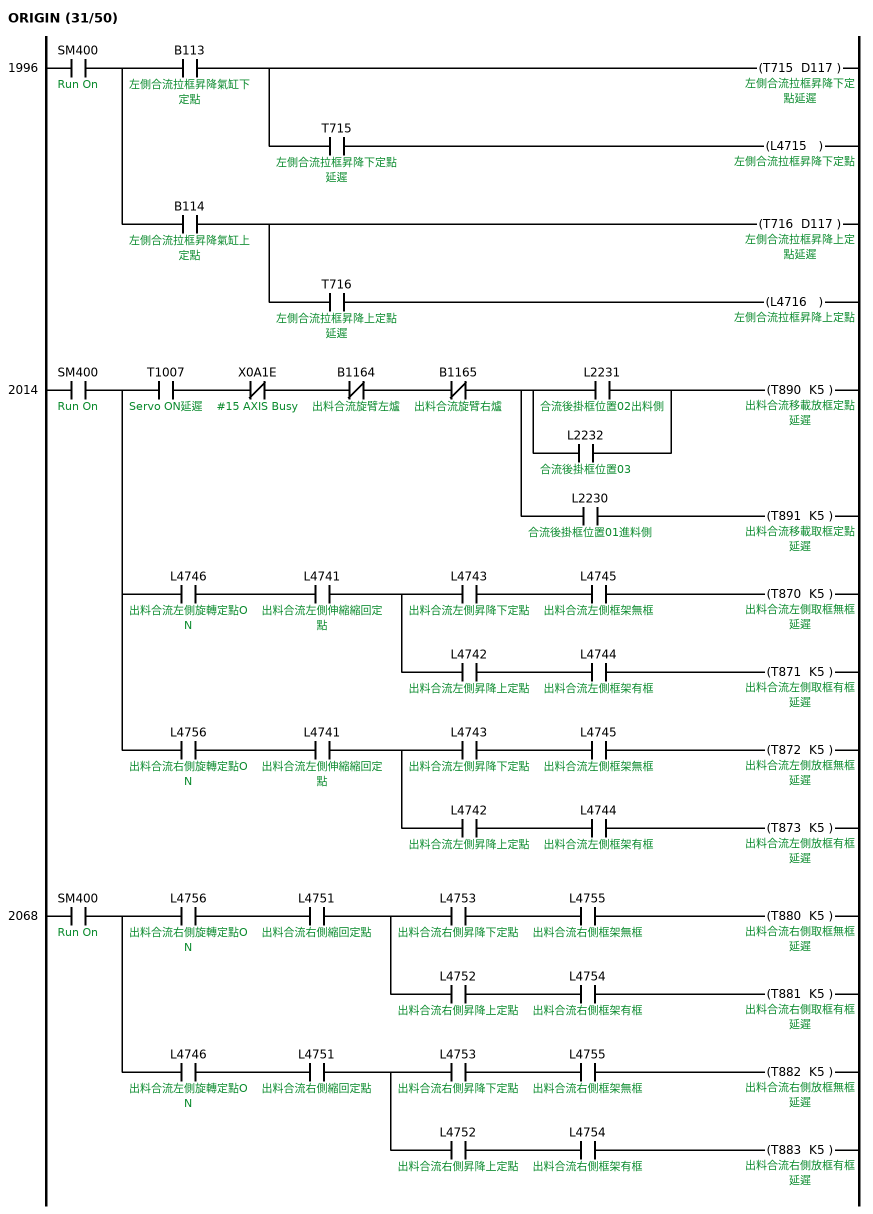
1996  LD      SM400  ; Run On
      MPS
      AND     B113  ; 左側合流拉框昇降氣缸下定點
      OUT     T715 D117  ; 左側合流拉框昇降下定點延遲
      AND     T715  ; 左側合流拉框昇降下定點延遲
      OUT     L4715  ; 左側合流拉框昇降下定點
      MPP
      AND     B114  ; 左側合流拉框昇降氣缸上定點
      OUT     T716 D117  ; 左側合流拉框昇降上定點延遲
      AND     T716  ; 左側合流拉框昇降上定點延遲
      OUT     L4716  ; 左側合流拉框昇降上定點
2014  LD      SM400  ; Run On
      MPS
      AND     T1007  ; Servo ON延遲
      ANI     X0A1E  ; #15 AXIS Busy
      ANI     B1164  ; 出料合流旋臂左爐
      ANI     B1165  ; 出料合流旋臂右爐
      MPS
      LD      L2231  ; 合流後掛框位置02出料側
      OR      L2232  ; 合流後掛框位置03
      ANB
      OUT     T890 K5  ; 出料合流移載放框定點延遲
      MPP
      AND     L2230  ; 合流後掛框位置01進料側
      OUT     T891 K5  ; 出料合流移載取框定點延遲
      MRD
      AND     L4746  ; 出料合流左側旋轉定點ON
      AND     L4741  ; 出料合流左側伸縮縮回定點
      MPS
      AND     L4743  ; 出料合流左側昇降下定點
      AND     L4745  ; 出料合流左側框架無框
      OUT     T870 K5  ; 出料合流左側取框無框延遲
      MPP
      AND     L4742  ; 出料合流左側昇降上定點
      AND     L4744  ; 出料合流左側框架有框
      OUT     T871 K5  ; 出料合流左側取框有框延遲
      MPP
      AND     L4756  ; 出料合流右側旋轉定點ON
      AND     L4741  ; 出料合流左側伸縮縮回定點
      MPS
      AND     L4743  ; 出料合流左側昇降下定點
      AND     L4745  ; 出料合流左側框架無框
      OUT     T872 K5  ; 出料合流左側放框無框延遲
      MPP
      AND     L4742  ; 出料合流左側昇降上定點
      AND     L4744  ; 出料合流左側框架有框
      OUT     T873 K5  ; 出料合流左側放框有框延遲
2068  LD      SM400  ; Run On
      MPS
      AND     L4756  ; 出料合流右側旋轉定點ON
      AND     L4751  ; 出料合流右側縮回定點
      MPS
      AND     L4753  ; 出料合流右側昇降下定點
      AND     L4755  ; 出料合流右側框架無框
      OUT     T880 K5  ; 出料合流右側取框無框延遲
      MPP
      AND     L4752  ; 出料合流右側昇降上定點
      AND     L4754  ; 出料合流右側框架有框
      OUT     T881 K5  ; 出料合流右側取框有框延遲
      MPP
      AND     L4746  ; 出料合流左側旋轉定點ON
      AND     L4751  ; 出料合流右側縮回定點
      MPS
      AND     L4753  ; 出料合流右側昇降下定點
      AND     L4755  ; 出料合流右側框架無框
      OUT     T882 K5  ; 出料合流右側放框無框延遲
      MPP
      AND     L4752  ; 出料合流右側昇降上定點
      AND     L4754  ; 出料合流右側框架有框
      OUT     T883 K5  ; 出料合流右側放框有框延遲
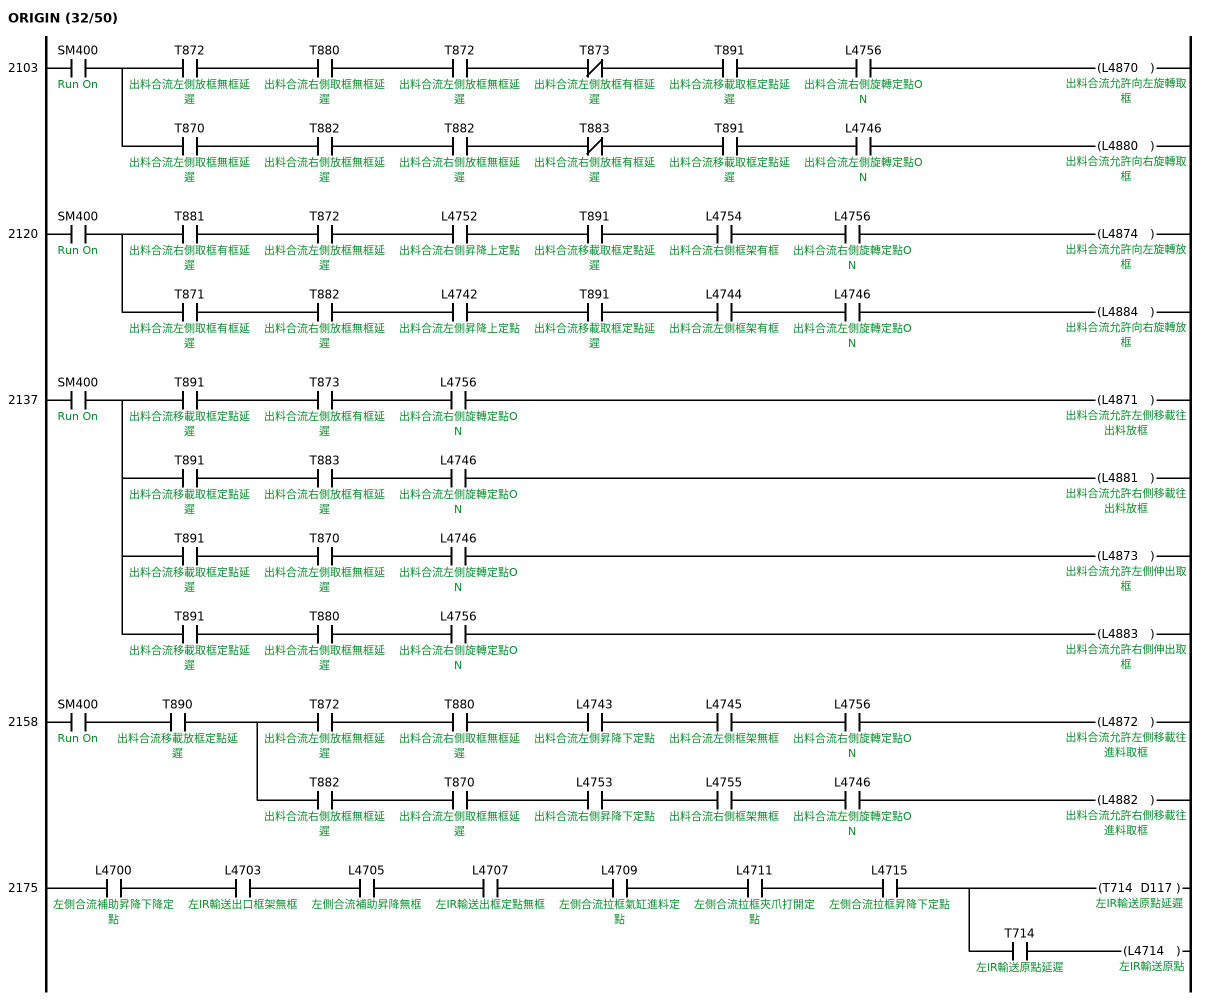
2103  LD      SM400  ; Run On
      MPS
      AND     T872  ; 出料合流左側放框無框延遲
      AND     T880  ; 出料合流右側取框無框延遲
      AND     T872  ; 出料合流左側放框無框延遲
      ANI     T873  ; 出料合流左側放框有框延遲
      AND     T891  ; 出料合流移載取框定點延遲
      AND     L4756  ; 出料合流右側旋轉定點ON
      OUT     L4870  ; 出料合流允許向左旋轉取框
      MPP
      AND     T870  ; 出料合流左側取框無框延遲
      AND     T882  ; 出料合流右側放框無框延遲
      AND     T882  ; 出料合流右側放框無框延遲
      ANI     T883  ; 出料合流右側放框有框延遲
      AND     T891  ; 出料合流移載取框定點延遲
      AND     L4746  ; 出料合流左側旋轉定點ON
      OUT     L4880  ; 出料合流允許向右旋轉取框
2120  LD      SM400  ; Run On
      MPS
      AND     T881  ; 出料合流右側取框有框延遲
      AND     T872  ; 出料合流左側放框無框延遲
      AND     L4752  ; 出料合流右側昇降上定點
      AND     T891  ; 出料合流移載取框定點延遲
      AND     L4754  ; 出料合流右側框架有框
      AND     L4756  ; 出料合流右側旋轉定點ON
      OUT     L4874  ; 出料合流允許向左旋轉放框
      MPP
      AND     T871  ; 出料合流左側取框有框延遲
      AND     T882  ; 出料合流右側放框無框延遲
      AND     L4742  ; 出料合流左側昇降上定點
      AND     T891  ; 出料合流移載取框定點延遲
      AND     L4744  ; 出料合流左側框架有框
      AND     L4746  ; 出料合流左側旋轉定點ON
      OUT     L4884  ; 出料合流允許向右旋轉放框
2137  LD      SM400  ; Run On
      MPS
      AND     T891  ; 出料合流移載取框定點延遲
      AND     T873  ; 出料合流左側放框有框延遲
      AND     L4756  ; 出料合流右側旋轉定點ON
      OUT     L4871  ; 出料合流允許左側移載往  出料放框
      MRD
      AND     T891  ; 出料合流移載取框定點延遲
      AND     T883  ; 出料合流右側放框有框延遲
      AND     L4746  ; 出料合流左側旋轉定點ON
      OUT     L4881  ; 出料合流允許右側移載往  出料放框
      MRD
      AND     T891  ; 出料合流移載取框定點延遲
      AND     T870  ; 出料合流左側取框無框延遲
      AND     L4746  ; 出料合流左側旋轉定點ON
      OUT     L4873  ; 出料合流允許左側伸出取框
      MPP
      AND     T891  ; 出料合流移載取框定點延遲
      AND     T880  ; 出料合流右側取框無框延遲
      AND     L4756  ; 出料合流右側旋轉定點ON
      OUT     L4883  ; 出料合流允許右側伸出取框
2158  LD      SM400  ; Run On
      AND     T890  ; 出料合流移載放框定點延遲
      MPS
      AND     T872  ; 出料合流左側放框無框延遲
      AND     T880  ; 出料合流右側取框無框延遲
      AND     L4743  ; 出料合流左側昇降下定點
      AND     L4745  ; 出料合流左側框架無框
      AND     L4756  ; 出料合流右側旋轉定點ON
      OUT     L4872  ; 出料合流允許左側移載往  進料取框
      MPP
      AND     T882  ; 出料合流右側放框無框延遲
      AND     T870  ; 出料合流左側取框無框延遲
      AND     L4753  ; 出料合流右側昇降下定點
      AND     L4755  ; 出料合流右側框架無框
      AND     L4746  ; 出料合流左側旋轉定點ON
      OUT     L4882  ; 出料合流允許右側移載往  進料取框
2175  LD      L4700  ; 左側合流補助昇降下降定點
      AND     L4703  ; 左IR輸送出口框架無框
      AND     L4705  ; 左側合流補助昇降無框
      AND     L4707  ; 左IR輸送出框定點無框
      AND     L4709  ; 左側合流拉框氣缸進料定點
      AND     L4711  ; 左側合流拉框夾爪打開定點
      AND     L4715  ; 左側合流拉框昇降下定點
      OUT     T714 D117  ; 左IR輸送原點延遲
      AND     T714  ; 左IR輸送原點延遲
      OUT     L4714  ; 左IR輸送原點
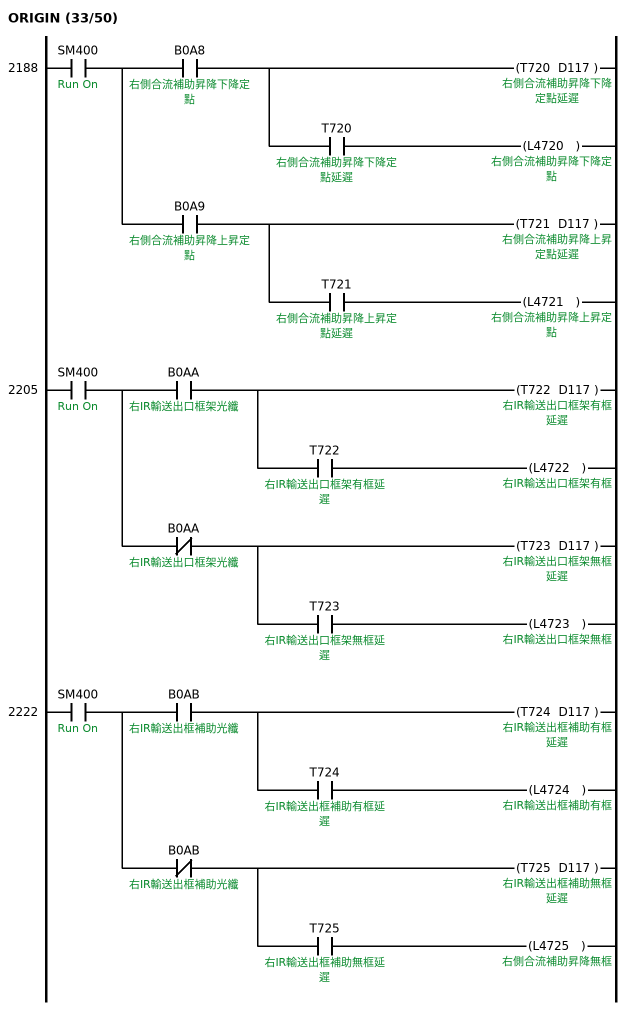
2188  LD      SM400  ; Run On
      MPS
      AND     B0A8  ; 右側合流補助昇降下降定點
      OUT     T720 D117  ; 右側合流補助昇降下降定點延遲
      AND     T720  ; 右側合流補助昇降下降定點延遲
      OUT     L4720  ; 右側合流補助昇降下降定點
      MPP
      AND     B0A9  ; 右側合流補助昇降上昇定點
      OUT     T721 D117  ; 右側合流補助昇降上昇定點延遲
      AND     T721  ; 右側合流補助昇降上昇定點延遲
      OUT     L4721  ; 右側合流補助昇降上昇定點
2205  LD      SM400  ; Run On
      MPS
      AND     B0AA  ; 右IR輸送出口框架光纖
      OUT     T722 D117  ; 右IR輸送出口框架有框延遲
      AND     T722  ; 右IR輸送出口框架有框延遲
      OUT     L4722  ; 右IR輸送出口框架有框
      MPP
      ANI     B0AA  ; 右IR輸送出口框架光纖
      OUT     T723 D117  ; 右IR輸送出口框架無框延遲
      AND     T723  ; 右IR輸送出口框架無框延遲
      OUT     L4723  ; 右IR輸送出口框架無框
2222  LD      SM400  ; Run On
      MPS
      AND     B0AB  ; 右IR輸送出框補助光纖
      OUT     T724 D117  ; 右IR輸送出框補助有框延遲
      AND     T724  ; 右IR輸送出框補助有框延遲
      OUT     L4724  ; 右IR輸送出框補助有框
      MPP
      ANI     B0AB  ; 右IR輸送出框補助光纖
      OUT     T725 D117  ; 右IR輸送出框補助無框延遲
      AND     T725  ; 右IR輸送出框補助無框延遲
      OUT     L4725  ; 右側合流補助昇降無框
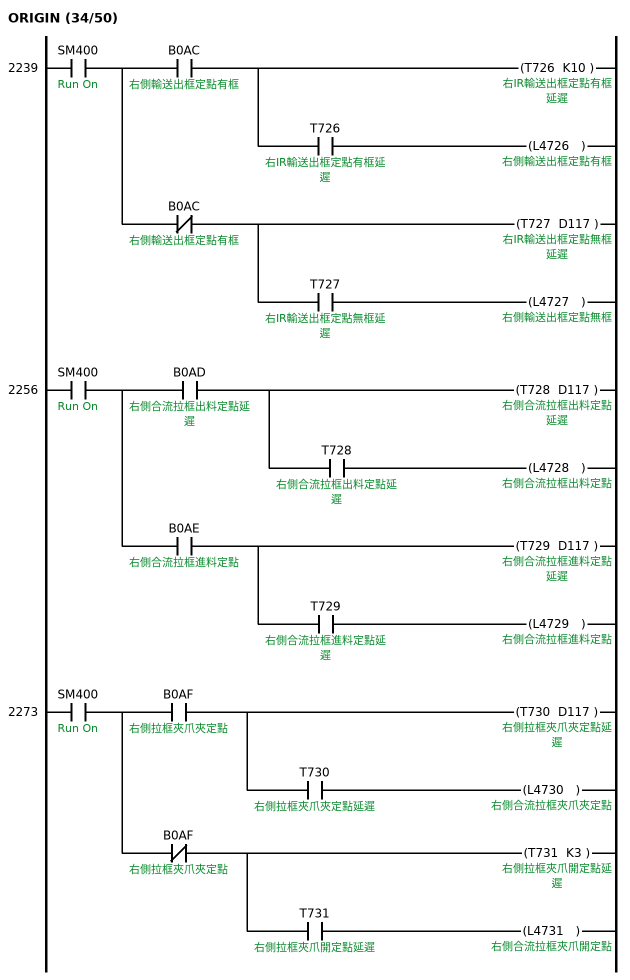
2239  LD      SM400  ; Run On
      MPS
      AND     B0AC  ; 右側輸送出框定點有框
      OUT     T726 K10  ; 右IR輸送出框定點有框延遲
      AND     T726  ; 右IR輸送出框定點有框延遲
      OUT     L4726  ; 右側輸送出框定點有框
      MPP
      ANI     B0AC  ; 右側輸送出框定點有框
      OUT     T727 D117  ; 右IR輸送出框定點無框延遲
      AND     T727  ; 右IR輸送出框定點無框延遲
      OUT     L4727  ; 右側輸送出框定點無框
2256  LD      SM400  ; Run On
      MPS
      AND     B0AD  ; 右側合流拉框出料定點延遲
      OUT     T728 D117  ; 右側合流拉框出料定點延遲
      AND     T728  ; 右側合流拉框出料定點延遲
      OUT     L4728  ; 右側合流拉框出料定點
      MPP
      AND     B0AE  ; 右側合流拉框進料定點
      OUT     T729 D117  ; 右側合流拉框進料定點延遲
      AND     T729  ; 右側合流拉框進料定點延遲
      OUT     L4729  ; 右側合流拉框進料定點
2273  LD      SM400  ; Run On
      MPS
      AND     B0AF  ; 右側拉框夾爪夾定點
      OUT     T730 D117  ; 右側拉框夾爪夾定點延遲
      AND     T730  ; 右側拉框夾爪夾定點延遲
      OUT     L4730  ; 右側合流拉框夾爪夾定點
      MPP
      ANI     B0AF  ; 右側拉框夾爪夾定點
      OUT     T731 K3  ; 右側拉框夾爪開定點延遲
      AND     T731  ; 右側拉框夾爪開定點延遲
      OUT     L4731  ; 右側合流拉框夾爪開定點
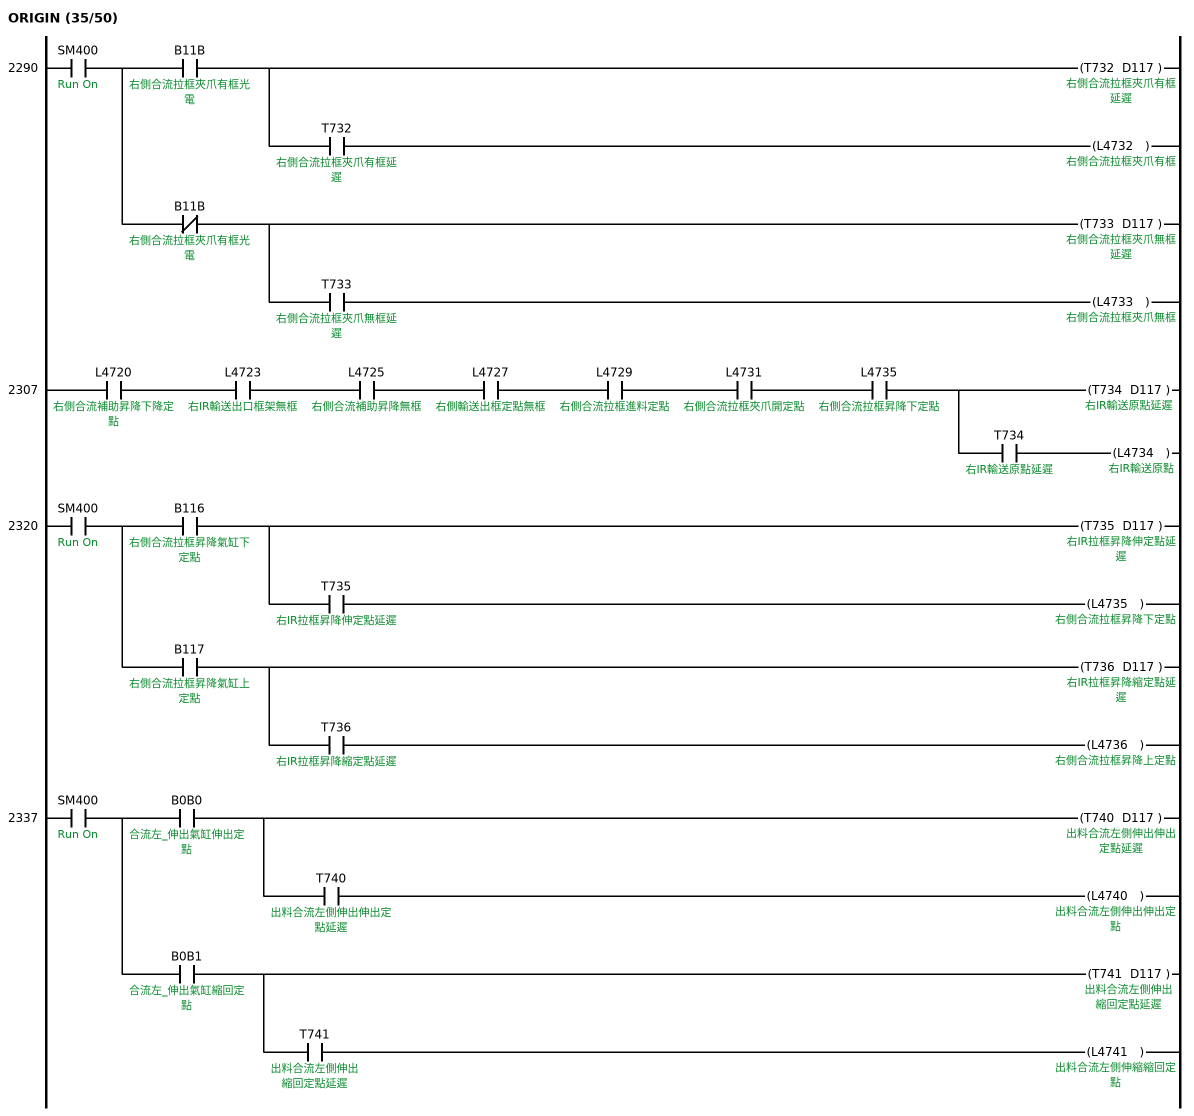
2290  LD      SM400  ; Run On
      MPS
      AND     B11B  ; 右側合流拉框夾爪有框光電
      OUT     T732 D117  ; 右側合流拉框夾爪有框延遲
      AND     T732  ; 右側合流拉框夾爪有框延遲
      OUT     L4732  ; 右側合流拉框夾爪有框
      MPP
      ANI     B11B  ; 右側合流拉框夾爪有框光電
      OUT     T733 D117  ; 右側合流拉框夾爪無框延遲
      AND     T733  ; 右側合流拉框夾爪無框延遲
      OUT     L4733  ; 右側合流拉框夾爪無框
2307  LD      L4720  ; 右側合流補助昇降下降定點
      AND     L4723  ; 右IR輸送出口框架無框
      AND     L4725  ; 右側合流補助昇降無框
      AND     L4727  ; 右側輸送出框定點無框
      AND     L4729  ; 右側合流拉框進料定點
      AND     L4731  ; 右側合流拉框夾爪開定點
      AND     L4735  ; 右側合流拉框昇降下定點
      OUT     T734 D117  ; 右IR輸送原點延遲
      AND     T734  ; 右IR輸送原點延遲
      OUT     L4734  ; 右IR輸送原點
2320  LD      SM400  ; Run On
      MPS
      AND     B116  ; 右側合流拉框昇降氣缸下定點
      OUT     T735 D117  ; 右IR拉框昇降伸定點延遲
      AND     T735  ; 右IR拉框昇降伸定點延遲
      OUT     L4735  ; 右側合流拉框昇降下定點
      MPP
      AND     B117  ; 右側合流拉框昇降氣缸上定點
      OUT     T736 D117  ; 右IR拉框昇降縮定點延遲
      AND     T736  ; 右IR拉框昇降縮定點延遲
      OUT     L4736  ; 右側合流拉框昇降上定點
2337  LD      SM400  ; Run On
      MPS
      AND     B0B0  ; 合流左_伸出氣缸伸出定點
      OUT     T740 D117  ; 出料合流左側伸出伸出定點延遲
      AND     T740  ; 出料合流左側伸出伸出定點延遲
      OUT     L4740  ; 出料合流左側伸出伸出定點
      MPP
      AND     B0B1  ; 合流左_伸出氣缸縮回定點
      OUT     T741 D117  ; 出料合流左側伸出 縮回定點延遲
      AND     T741  ; 出料合流左側伸出 縮回定點延遲
      OUT     L4741  ; 出料合流左側伸縮縮回定點
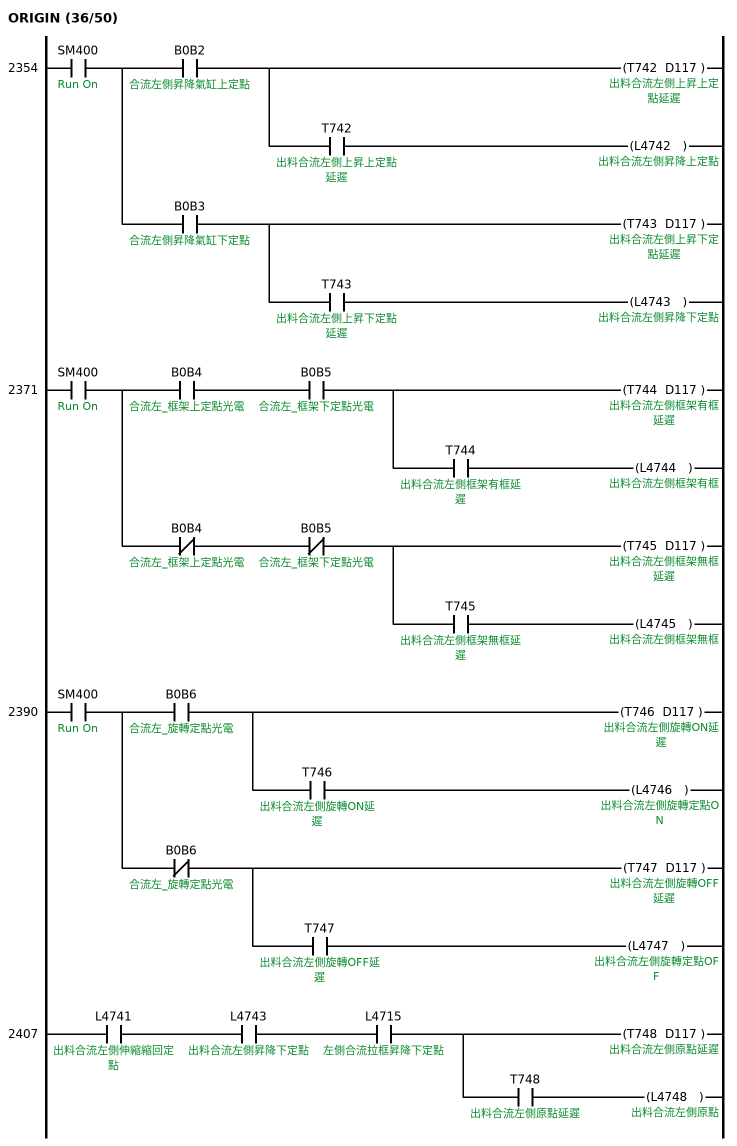
2354  LD      SM400  ; Run On
      MPS
      AND     B0B2  ; 合流左側昇降氣缸上定點
      OUT     T742 D117  ; 出料合流左側上昇上定點延遲
      AND     T742  ; 出料合流左側上昇上定點延遲
      OUT     L4742  ; 出料合流左側昇降上定點
      MPP
      AND     B0B3  ; 合流左側昇降氣缸下定點
      OUT     T743 D117  ; 出料合流左側上昇下定點延遲
      AND     T743  ; 出料合流左側上昇下定點延遲
      OUT     L4743  ; 出料合流左側昇降下定點
2371  LD      SM400  ; Run On
      MPS
      AND     B0B4  ; 合流左_框架上定點光電
      AND     B0B5  ; 合流左_框架下定點光電
      OUT     T744 D117  ; 出料合流左側框架有框延遲
      AND     T744  ; 出料合流左側框架有框延遲
      OUT     L4744  ; 出料合流左側框架有框
      MPP
      ANI     B0B4  ; 合流左_框架上定點光電
      ANI     B0B5  ; 合流左_框架下定點光電
      OUT     T745 D117  ; 出料合流左側框架無框延遲
      AND     T745  ; 出料合流左側框架無框延遲
      OUT     L4745  ; 出料合流左側框架無框
2390  LD      SM400  ; Run On
      MPS
      AND     B0B6  ; 合流左_旋轉定點光電
      OUT     T746 D117  ; 出料合流左側旋轉ON延遲
      AND     T746  ; 出料合流左側旋轉ON延遲
      OUT     L4746  ; 出料合流左側旋轉定點ON
      MPP
      ANI     B0B6  ; 合流左_旋轉定點光電
      OUT     T747 D117  ; 出料合流左側旋轉OFF延遲
      AND     T747  ; 出料合流左側旋轉OFF延遲
      OUT     L4747  ; 出料合流左側旋轉定點OFF
2407  LD      L4741  ; 出料合流左側伸縮縮回定點
      AND     L4743  ; 出料合流左側昇降下定點
      AND     L4715  ; 左側合流拉框昇降下定點
      OUT     T748 D117  ; 出料合流左側原點延遲
      AND     T748  ; 出料合流左側原點延遲
      OUT     L4748  ; 出料合流左側原點
